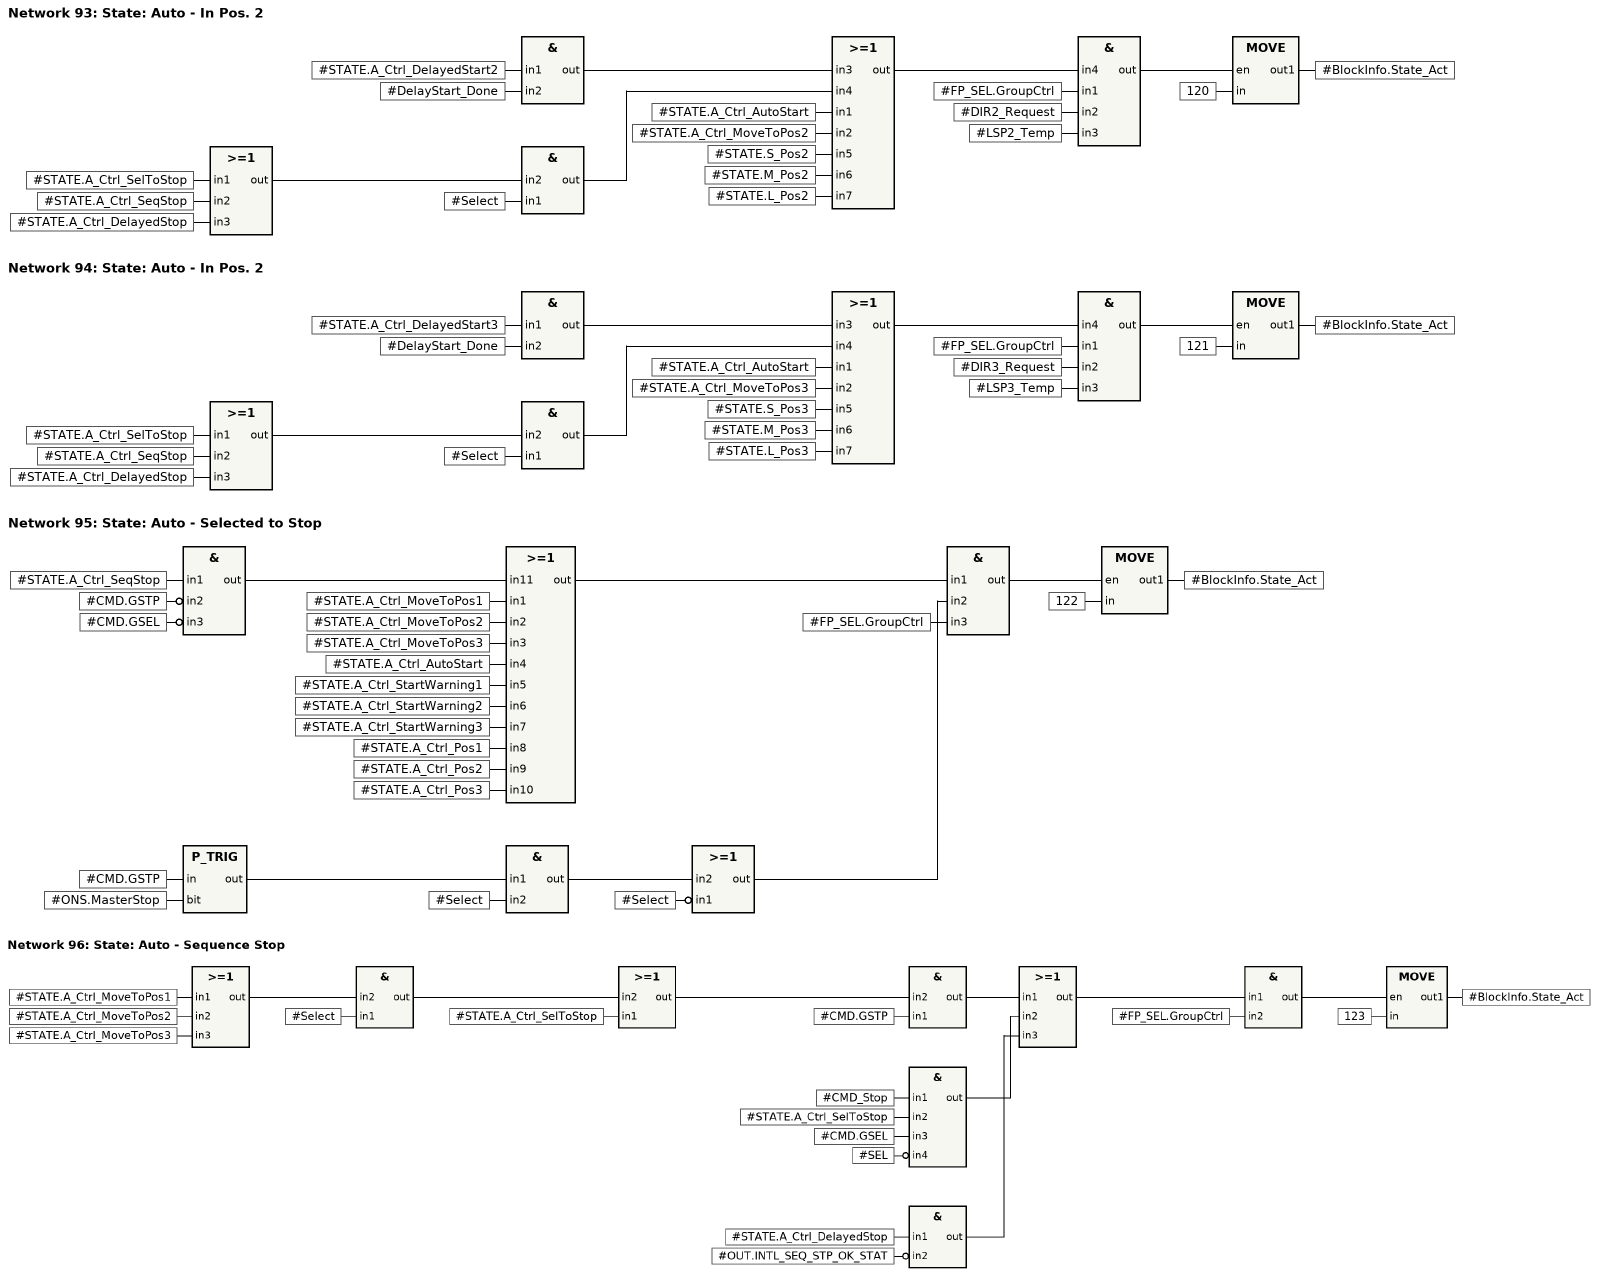
   IF ((#STATE.A_Ctrl_DelayedStart2 AND #DelayStart_Done) OR ((#STATE.A_Ctrl_SelToStop OR #STATE.A_Ctrl_SeqStop OR #STATE.A_Ctrl_DelayedStop) AND #Select) OR #STATE.A_Ctrl_AutoStart OR #STATE.A_Ctrl_MoveToPos2 OR #STATE.S_Pos2 OR #STATE.M_Pos2 OR #STATE.L_Pos2) AND #FP_SEL.GroupCtrl AND #DIR2_Request AND #LSP2_Temp THEN
       #BlockInfo.State_Act := 120;
   END_IF;
END_REGION

REGION Network 94: State: Auto - In Pos. 2
   IF ((#STATE.A_Ctrl_DelayedStart3 AND #DelayStart_Done) OR ((#STATE.A_Ctrl_SelToStop OR #STATE.A_Ctrl_SeqStop OR #STATE.A_Ctrl_DelayedStop) AND #Select) OR #STATE.A_Ctrl_AutoStart OR #STATE.A_Ctrl_MoveToPos3 OR #STATE.S_Pos3 OR #STATE.M_Pos3 OR #STATE.L_Pos3) AND #FP_SEL.GroupCtrl AND #DIR3_Request AND #LSP3_Temp THEN
       #BlockInfo.State_Act := 121;
   END_IF;
END_REGION

REGION Network 95: State: Auto - Selected to Stop
   // Build 004 - 11 Jul 2019 (EXTBOB) : GSEL and A_Ctrl_SeqStop with GSTP condition to move to Selected to Stop state from Seq stop state if group stop timer completes
   #_w1 := #CMD.GSTP AND NOT #ONS.MasterStop;   // rising edge
   #ONS.MasterStop := #CMD.GSTP;
   IF ((#STATE.A_Ctrl_SeqStop AND NOT #CMD.GSTP AND NOT #CMD.GSEL) OR #STATE.A_Ctrl_MoveToPos1 OR #STATE.A_Ctrl_MoveToPos2 OR #STATE.A_Ctrl_MoveToPos3 OR #STATE.A_Ctrl_AutoStart OR #STATE.A_Ctrl_StartWarning1 OR #STATE.A_Ctrl_StartWarning2 OR #STATE.A_Ctrl_StartWarning3 OR #STATE.A_Ctrl_Pos1 OR #STATE.A_Ctrl_Pos2 OR #STATE.A_Ctrl_Pos3) AND ((#_w1 AND #Select) OR NOT #Select) AND #FP_SEL.GroupCtrl THEN
       #BlockInfo.State_Act := 122;
   END_IF;
END_REGION

REGION Network 96: State: Auto - Sequence Stop
   IF (((((#STATE.A_Ctrl_MoveToPos1 OR #STATE.A_Ctrl_MoveToPos2 OR #STATE.A_Ctrl_MoveToPos3) AND #Select) OR #STATE.A_Ctrl_SelToStop) AND #CMD.GSTP) OR (#CMD_Stop AND #STATE.A_Ctrl_SelToStop AND #CMD.GSEL AND NOT #SEL) OR (#STATE.A_Ctrl_DelayedStop AND NOT #OUT.INTL_SEQ_STP_OK_STAT)) AND #FP_SEL.GroupCtrl THEN
       #BlockInfo.State_Act := 123;
   END_IF;
END_REGION

REGION Network 97: State: Auto - Delayed Stop
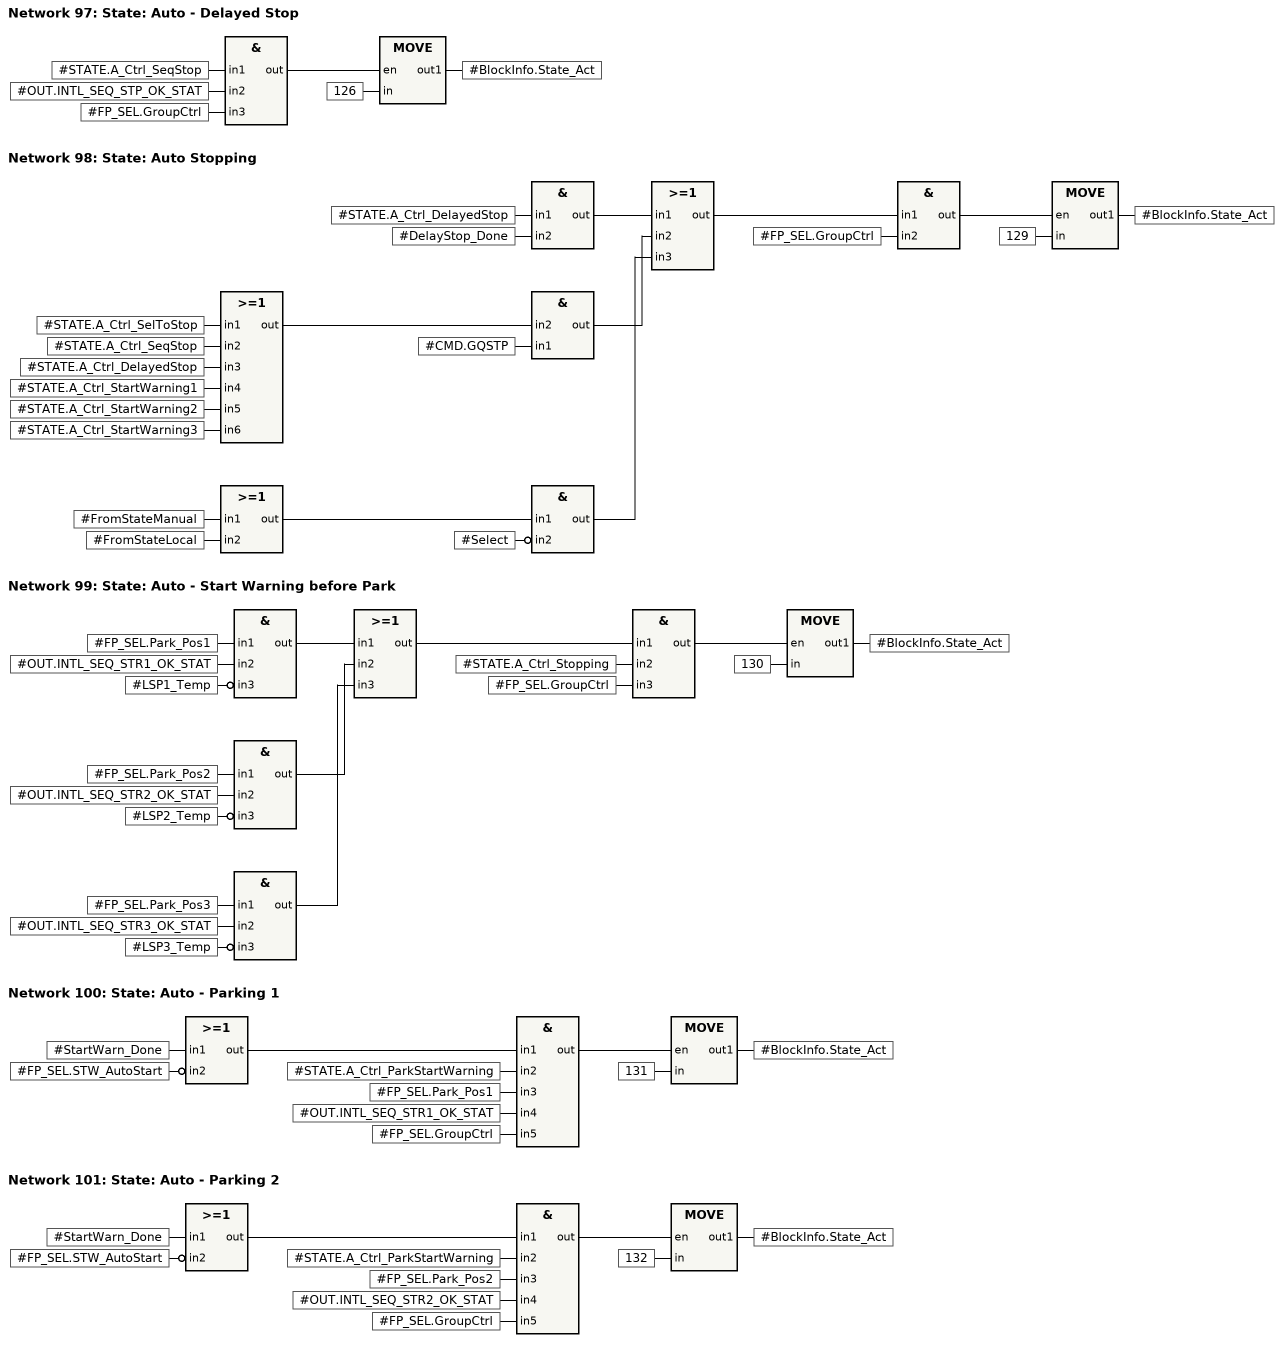
   IF #STATE.A_Ctrl_SeqStop AND #OUT.INTL_SEQ_STP_OK_STAT AND #FP_SEL.GroupCtrl THEN
       #BlockInfo.State_Act := 126;
   END_IF;
END_REGION

REGION Network 98: State: Auto Stopping
   IF ((#STATE.A_Ctrl_DelayedStop AND #DelayStop_Done) OR ((#STATE.A_Ctrl_SelToStop OR #STATE.A_Ctrl_SeqStop OR #STATE.A_Ctrl_DelayedStop OR #STATE.A_Ctrl_StartWarning1 OR #STATE.A_Ctrl_StartWarning2 OR #STATE.A_Ctrl_StartWarning3) AND #CMD.GQSTP) OR ((#FromStateManual OR #FromStateLocal) AND NOT #Select)) AND #FP_SEL.GroupCtrl THEN
       #BlockInfo.State_Act := 129;
   END_IF;
END_REGION

REGION Network 99: State: Auto - Start Warning before Park
   IF ((#FP_SEL.Park_Pos1 AND #OUT.INTL_SEQ_STR1_OK_STAT AND NOT #LSP1_Temp) OR (#FP_SEL.Park_Pos2 AND #OUT.INTL_SEQ_STR2_OK_STAT AND NOT #LSP2_Temp) OR (#FP_SEL.Park_Pos3 AND #OUT.INTL_SEQ_STR3_OK_STAT AND NOT #LSP3_Temp)) AND #STATE.A_Ctrl_Stopping AND #FP_SEL.GroupCtrl THEN
       #BlockInfo.State_Act := 130;
   END_IF;
END_REGION

REGION Network 100: State: Auto - Parking 1
   IF (#StartWarn_Done OR NOT #FP_SEL.STW_AutoStart) AND #STATE.A_Ctrl_ParkStartWarning AND #FP_SEL.Park_Pos1 AND #OUT.INTL_SEQ_STR1_OK_STAT AND #FP_SEL.GroupCtrl THEN
       #BlockInfo.State_Act := 131;
   END_IF;
END_REGION

REGION Network 101: State: Auto - Parking 2
   IF (#StartWarn_Done OR NOT #FP_SEL.STW_AutoStart) AND #STATE.A_Ctrl_ParkStartWarning AND #FP_SEL.Park_Pos2 AND #OUT.INTL_SEQ_STR2_OK_STAT AND #FP_SEL.GroupCtrl THEN
       #BlockInfo.State_Act := 132;
   END_IF;
END_REGION

REGION Network 102: State: Auto - Parking 3
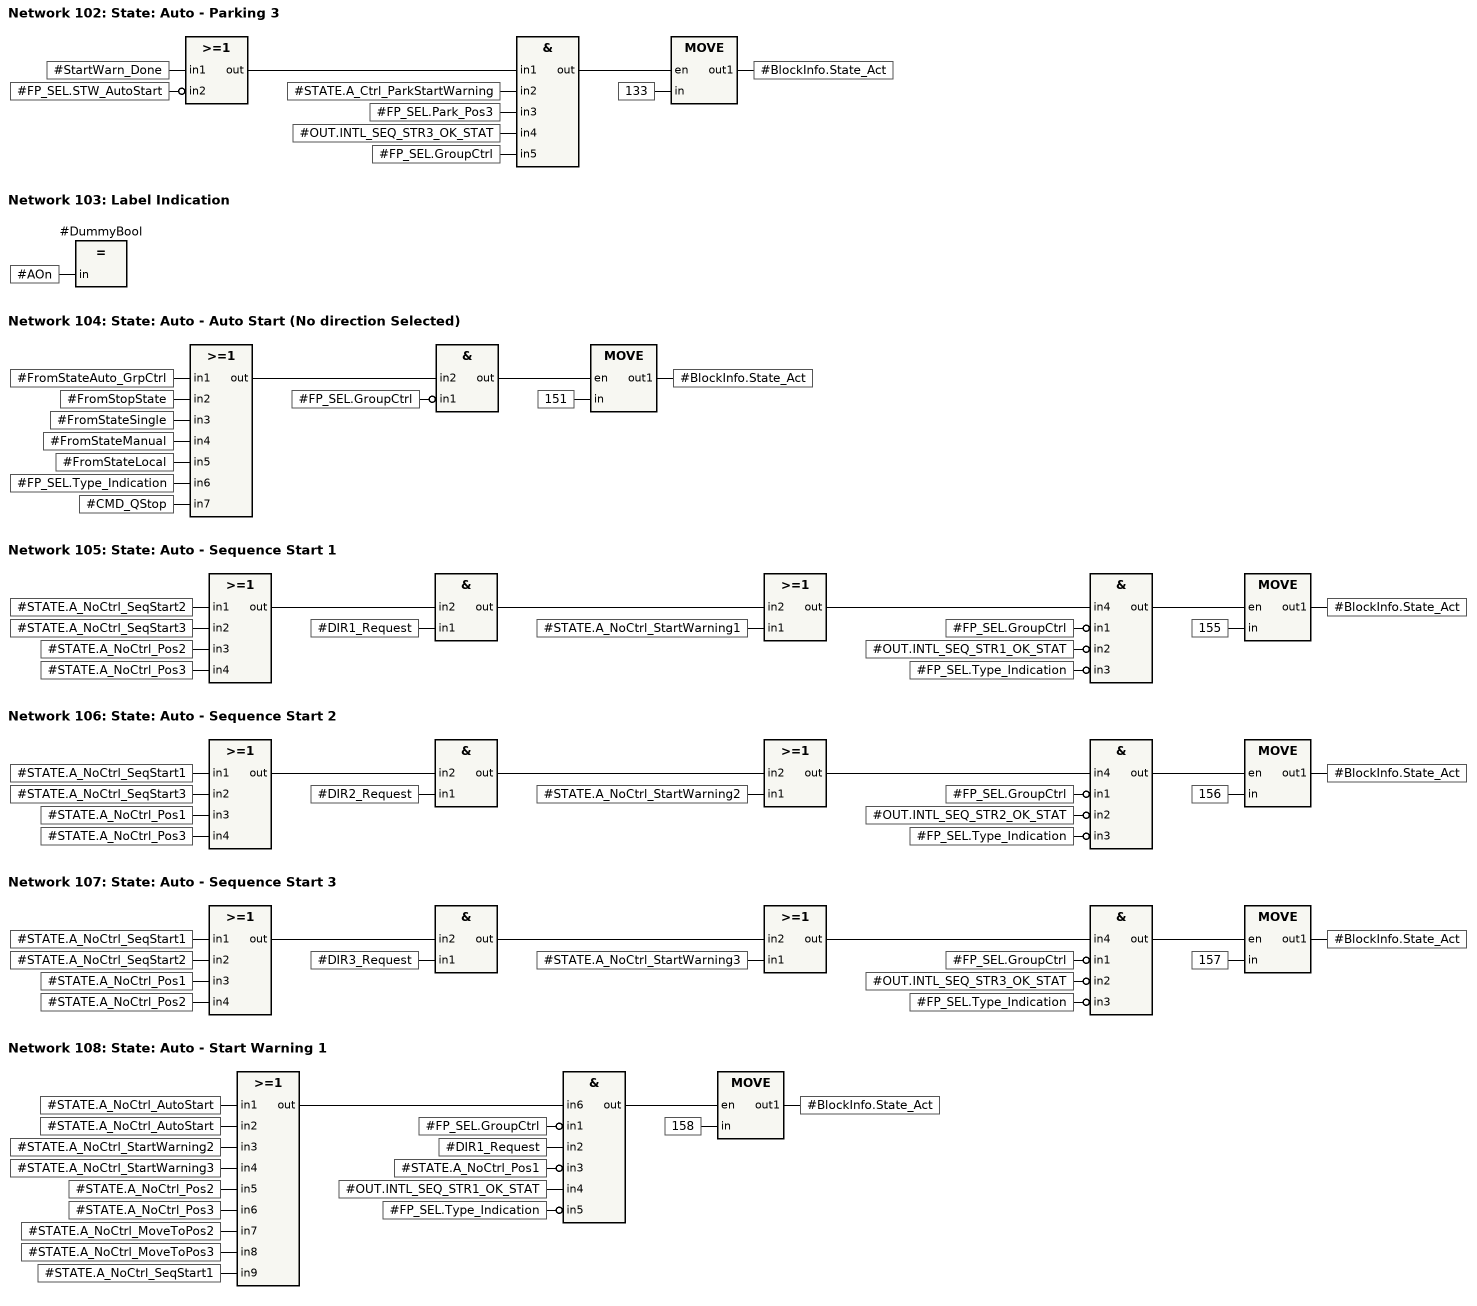
   IF (#StartWarn_Done OR NOT #FP_SEL.STW_AutoStart) AND #STATE.A_Ctrl_ParkStartWarning AND #FP_SEL.Park_Pos3 AND #OUT.INTL_SEQ_STR3_OK_STAT AND #FP_SEL.GroupCtrl THEN
       #BlockInfo.State_Act := 133;
   END_IF;
END_REGION

REGION Network 103: Label Indication
   INDC:
   #DummyBool := #AOn;
END_REGION

REGION Network 104: State: Auto - Auto Start (No direction Selected)
   IF (#FromStateAuto_GrpCtrl OR #FromStopState OR #FromStateSingle OR #FromStateManual OR #FromStateLocal OR #FP_SEL.Type_Indication OR #CMD_QStop) AND NOT #FP_SEL.GroupCtrl THEN
       #BlockInfo.State_Act := 151;
   END_IF;
END_REGION

REGION Network 105: State: Auto - Sequence Start 1
   IF (((#STATE.A_NoCtrl_SeqStart2 OR #STATE.A_NoCtrl_SeqStart3 OR #STATE.A_NoCtrl_Pos2 OR #STATE.A_NoCtrl_Pos3) AND #DIR1_Request) OR #STATE.A_NoCtrl_StartWarning1) AND NOT #FP_SEL.GroupCtrl AND NOT #OUT.INTL_SEQ_STR1_OK_STAT AND NOT #FP_SEL.Type_Indication THEN
       #BlockInfo.State_Act := 155;
   END_IF;
END_REGION

REGION Network 106: State: Auto - Sequence Start 2
   IF (((#STATE.A_NoCtrl_SeqStart1 OR #STATE.A_NoCtrl_SeqStart3 OR #STATE.A_NoCtrl_Pos1 OR #STATE.A_NoCtrl_Pos3) AND #DIR2_Request) OR #STATE.A_NoCtrl_StartWarning2) AND NOT #FP_SEL.GroupCtrl AND NOT #OUT.INTL_SEQ_STR2_OK_STAT AND NOT #FP_SEL.Type_Indication THEN
       #BlockInfo.State_Act := 156;
   END_IF;
END_REGION

REGION Network 107: State: Auto - Sequence Start 3
   IF (((#STATE.A_NoCtrl_SeqStart1 OR #STATE.A_NoCtrl_SeqStart2 OR #STATE.A_NoCtrl_Pos1 OR #STATE.A_NoCtrl_Pos2) AND #DIR3_Request) OR #STATE.A_NoCtrl_StartWarning3) AND NOT #FP_SEL.GroupCtrl AND NOT #OUT.INTL_SEQ_STR3_OK_STAT AND NOT #FP_SEL.Type_Indication THEN
       #BlockInfo.State_Act := 157;
   END_IF;
END_REGION

REGION Network 108: State: Auto - Start Warning 1
   IF (#STATE.A_NoCtrl_AutoStart OR #STATE.A_NoCtrl_AutoStart OR #STATE.A_NoCtrl_StartWarning2 OR #STATE.A_NoCtrl_StartWarning3 OR #STATE.A_NoCtrl_Pos2 OR #STATE.A_NoCtrl_Pos3 OR #STATE.A_NoCtrl_MoveToPos2 OR #STATE.A_NoCtrl_MoveToPos3 OR #STATE.A_NoCtrl_SeqStart1) AND NOT #FP_SEL.GroupCtrl AND #DIR1_Request AND NOT #STATE.A_NoCtrl_Pos1 AND #OUT.INTL_SEQ_STR1_OK_STAT AND NOT #FP_SEL.Type_Indication THEN
       #BlockInfo.State_Act := 158;
   END_IF;
END_REGION

REGION Network 109: State: Auto - Start Warning 2
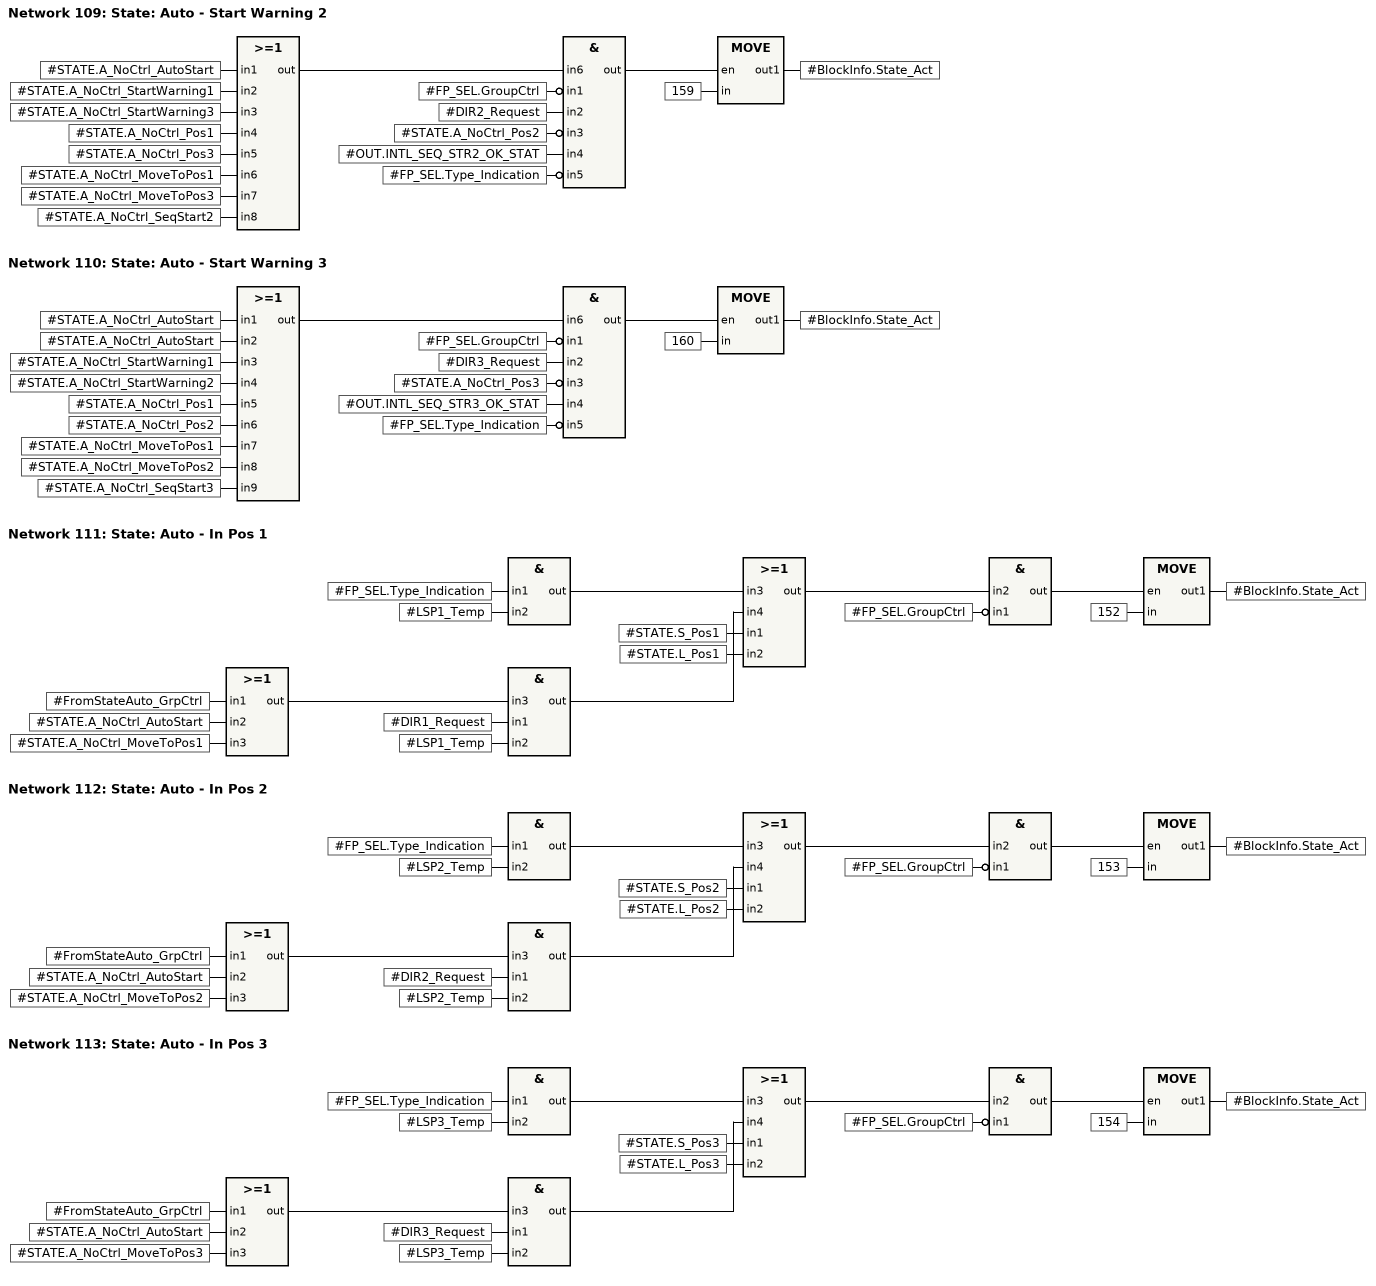
   IF (#STATE.A_NoCtrl_AutoStart OR #STATE.A_NoCtrl_StartWarning1 OR #STATE.A_NoCtrl_StartWarning3 OR #STATE.A_NoCtrl_Pos1 OR #STATE.A_NoCtrl_Pos3 OR #STATE.A_NoCtrl_MoveToPos1 OR #STATE.A_NoCtrl_MoveToPos3 OR #STATE.A_NoCtrl_SeqStart2) AND NOT #FP_SEL.GroupCtrl AND #DIR2_Request AND NOT #STATE.A_NoCtrl_Pos2 AND #OUT.INTL_SEQ_STR2_OK_STAT AND NOT #FP_SEL.Type_Indication THEN
       #BlockInfo.State_Act := 159;
   END_IF;
END_REGION

REGION Network 110: State: Auto - Start Warning 3
   IF (#STATE.A_NoCtrl_AutoStart OR #STATE.A_NoCtrl_AutoStart OR #STATE.A_NoCtrl_StartWarning1 OR #STATE.A_NoCtrl_StartWarning2 OR #STATE.A_NoCtrl_Pos1 OR #STATE.A_NoCtrl_Pos2 OR #STATE.A_NoCtrl_MoveToPos1 OR #STATE.A_NoCtrl_MoveToPos2 OR #STATE.A_NoCtrl_SeqStart3) AND NOT #FP_SEL.GroupCtrl AND #DIR3_Request AND NOT #STATE.A_NoCtrl_Pos3 AND #OUT.INTL_SEQ_STR3_OK_STAT AND NOT #FP_SEL.Type_Indication THEN
       #BlockInfo.State_Act := 160;
   END_IF;
END_REGION

REGION Network 111: State: Auto - In Pos 1
   IF ((#FP_SEL.Type_Indication AND #LSP1_Temp) OR ((#FromStateAuto_GrpCtrl OR #STATE.A_NoCtrl_AutoStart OR #STATE.A_NoCtrl_MoveToPos1) AND #DIR1_Request AND #LSP1_Temp) OR #STATE.S_Pos1 OR #STATE.L_Pos1) AND NOT #FP_SEL.GroupCtrl THEN
       #BlockInfo.State_Act := 152;
   END_IF;
END_REGION

REGION Network 112: State: Auto - In Pos 2
   IF ((#FP_SEL.Type_Indication AND #LSP2_Temp) OR ((#FromStateAuto_GrpCtrl OR #STATE.A_NoCtrl_AutoStart OR #STATE.A_NoCtrl_MoveToPos2) AND #DIR2_Request AND #LSP2_Temp) OR #STATE.S_Pos2 OR #STATE.L_Pos2) AND NOT #FP_SEL.GroupCtrl THEN
       #BlockInfo.State_Act := 153;
   END_IF;
END_REGION

REGION Network 113: State: Auto - In Pos 3
   IF ((#FP_SEL.Type_Indication AND #LSP3_Temp) OR ((#FromStateAuto_GrpCtrl OR #STATE.A_NoCtrl_AutoStart OR #STATE.A_NoCtrl_MoveToPos3) AND #DIR3_Request AND #LSP3_Temp) OR #STATE.S_Pos3 OR #STATE.L_Pos3) AND NOT #FP_SEL.GroupCtrl THEN
       #BlockInfo.State_Act := 154;
   END_IF;
END_REGION

REGION Network 114: State: Auto - Running 1
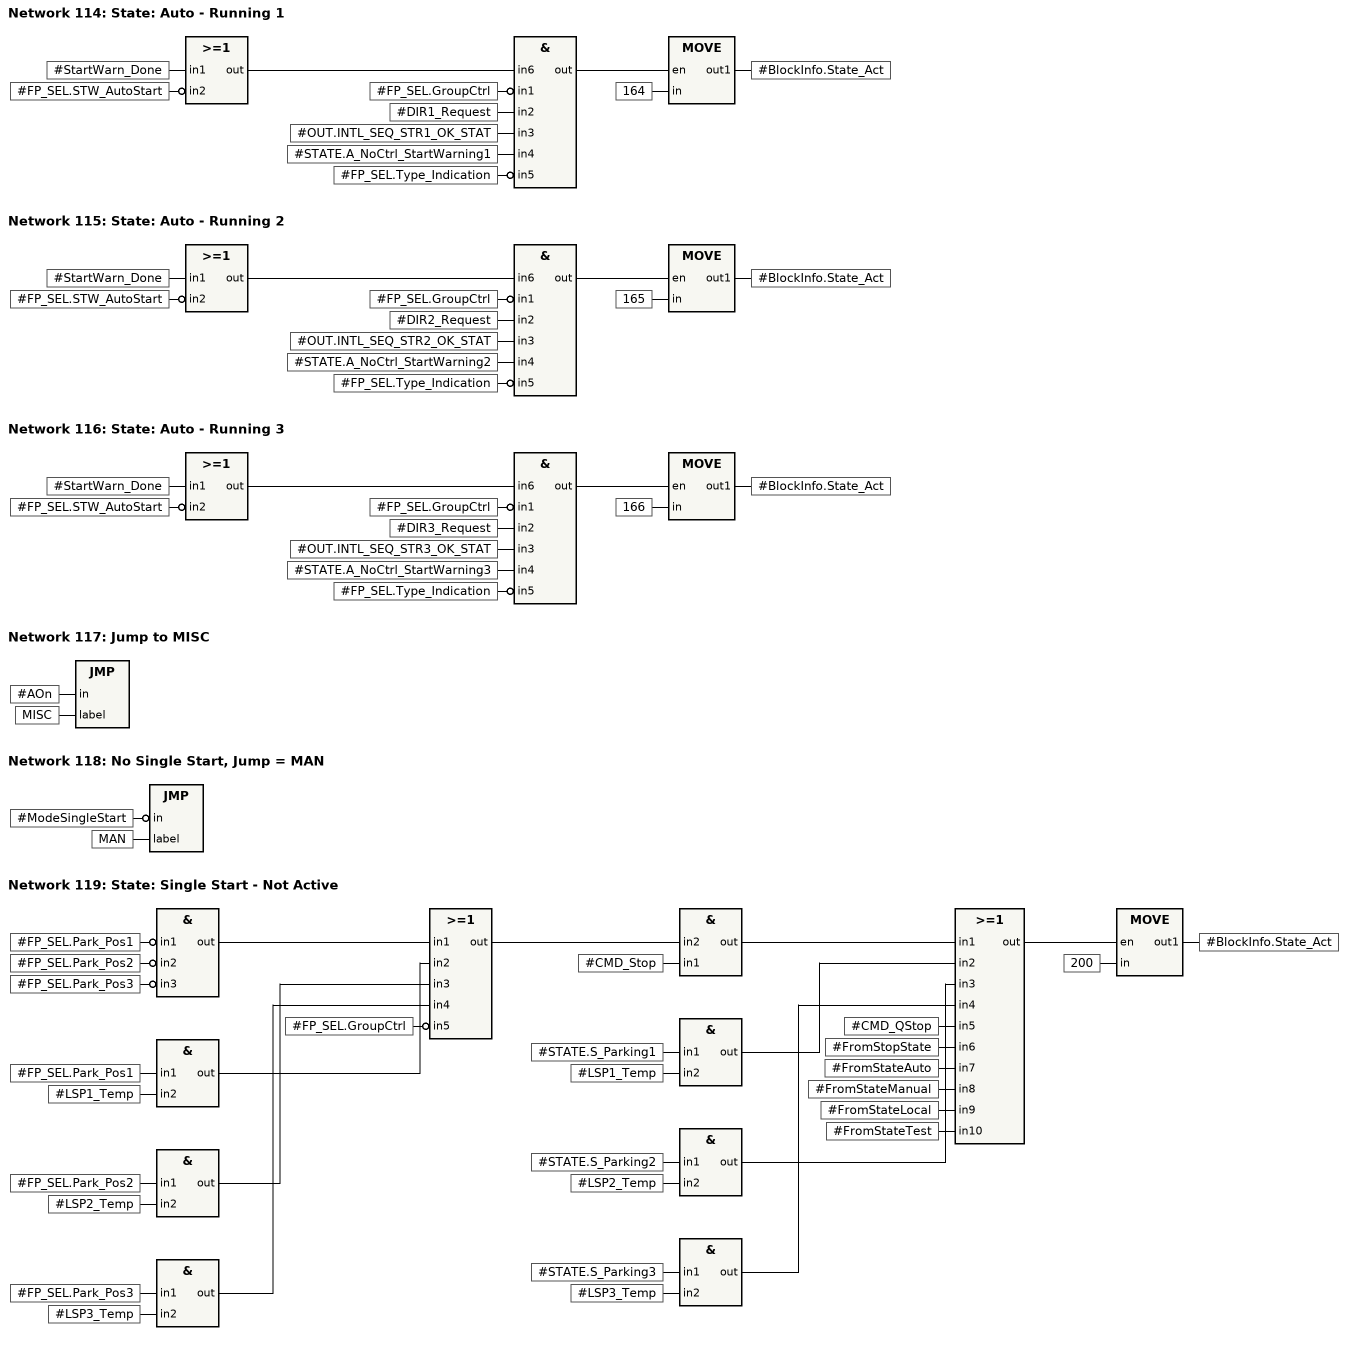
   IF (#StartWarn_Done OR NOT #FP_SEL.STW_AutoStart) AND NOT #FP_SEL.GroupCtrl AND #DIR1_Request AND #OUT.INTL_SEQ_STR1_OK_STAT AND #STATE.A_NoCtrl_StartWarning1 AND NOT #FP_SEL.Type_Indication THEN
       #BlockInfo.State_Act := 164;
   END_IF;
END_REGION

REGION Network 115: State: Auto - Running 2
   IF (#StartWarn_Done OR NOT #FP_SEL.STW_AutoStart) AND NOT #FP_SEL.GroupCtrl AND #DIR2_Request AND #OUT.INTL_SEQ_STR2_OK_STAT AND #STATE.A_NoCtrl_StartWarning2 AND NOT #FP_SEL.Type_Indication THEN
       #BlockInfo.State_Act := 165;
   END_IF;
END_REGION

REGION Network 116: State: Auto - Running 3
   IF (#StartWarn_Done OR NOT #FP_SEL.STW_AutoStart) AND NOT #FP_SEL.GroupCtrl AND #DIR3_Request AND #OUT.INTL_SEQ_STR3_OK_STAT AND #STATE.A_NoCtrl_StartWarning3 AND NOT #FP_SEL.Type_Indication THEN
       #BlockInfo.State_Act := 166;
   END_IF;
END_REGION

REGION Network 117: Jump to MISC
   IF #AOn THEN GOTO MISC; END_IF;
END_REGION

REGION Network 118: No Single Start, Jump = MAN
   SS1:
   IF NOT #ModeSingleStart THEN GOTO MAN; END_IF;
END_REGION

REGION Network 119: State: Single Start - Not Active
   IF (((NOT #FP_SEL.Park_Pos1 AND NOT #FP_SEL.Park_Pos2 AND NOT #FP_SEL.Park_Pos3) OR (#FP_SEL.Park_Pos1 AND #LSP1_Temp) OR (#FP_SEL.Park_Pos2 AND #LSP2_Temp) OR (#FP_SEL.Park_Pos3 AND #LSP3_Temp) OR NOT #FP_SEL.GroupCtrl) AND #CMD_Stop) OR (#STATE.S_Parking1 AND #LSP1_Temp) OR (#STATE.S_Parking2 AND #LSP2_Temp) OR (#STATE.S_Parking3 AND #LSP3_Temp) OR #CMD_QStop OR #FromStopState OR #FromStateAuto OR #FromStateManual OR #FromStateLocal OR #FromStateTest THEN
       #BlockInfo.State_Act := 200;
   END_IF;
END_REGION

REGION Network 120: State: Single Start - Start Warning 1
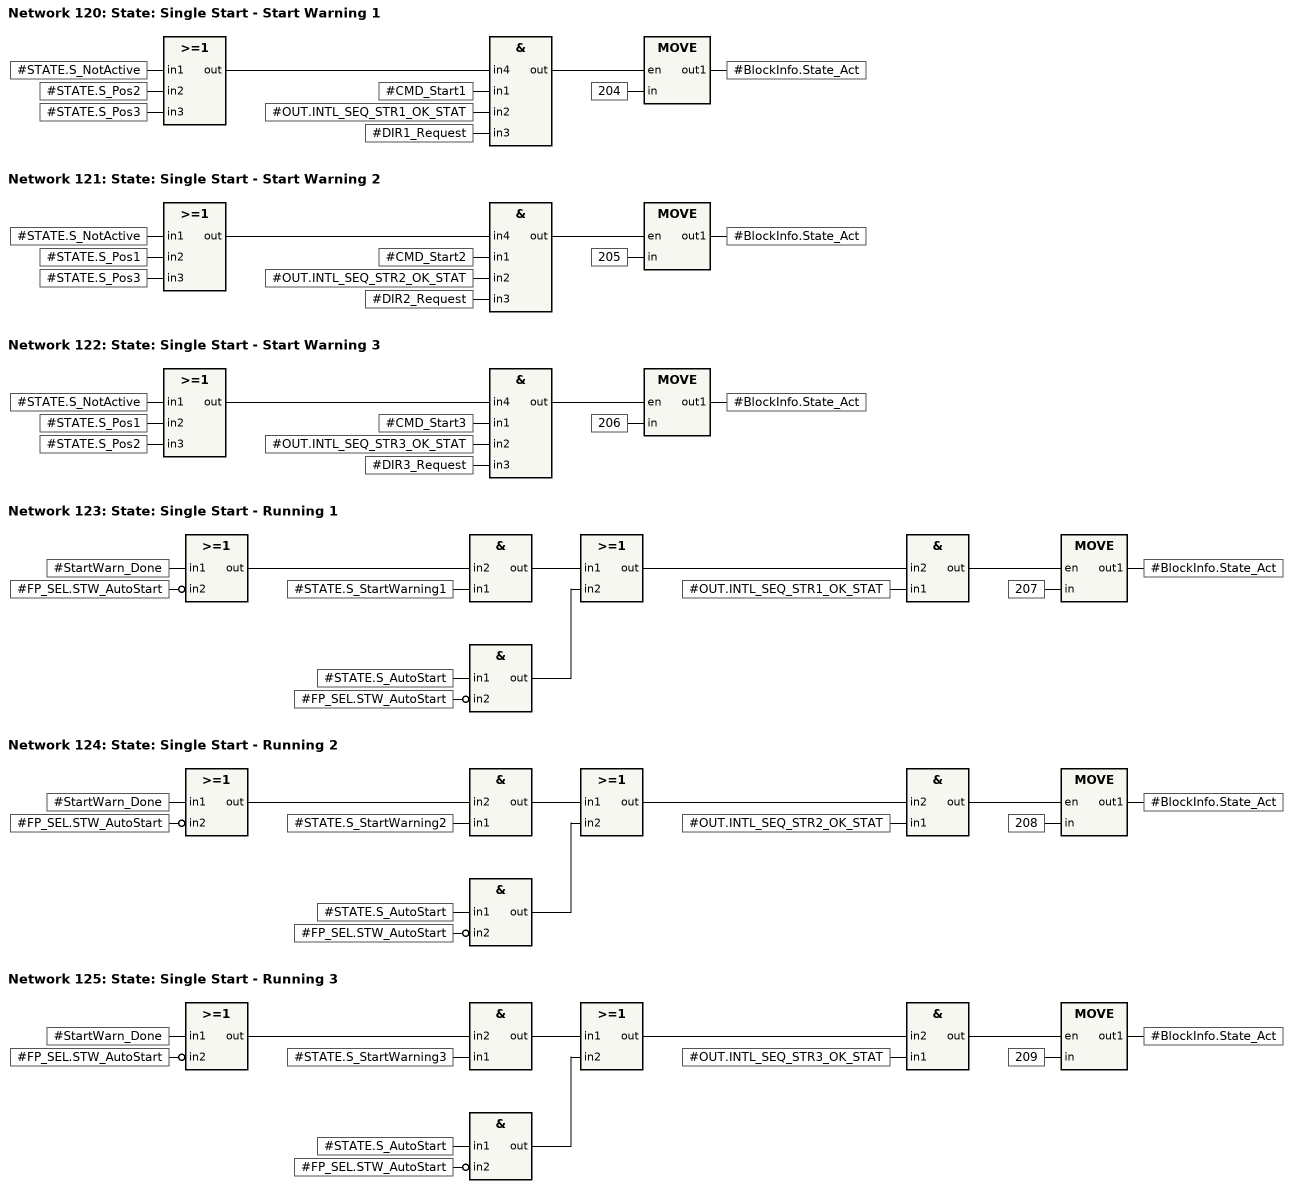
   IF (#STATE.S_NotActive OR #STATE.S_Pos2 OR #STATE.S_Pos3) AND #CMD_Start1 AND #OUT.INTL_SEQ_STR1_OK_STAT AND #DIR1_Request THEN
       #BlockInfo.State_Act := 204;
   END_IF;
END_REGION

REGION Network 121: State: Single Start - Start Warning 2
   IF (#STATE.S_NotActive OR #STATE.S_Pos1 OR #STATE.S_Pos3) AND #CMD_Start2 AND #OUT.INTL_SEQ_STR2_OK_STAT AND #DIR2_Request THEN
       #BlockInfo.State_Act := 205;
   END_IF;
END_REGION

REGION Network 122: State: Single Start - Start Warning 3
   IF (#STATE.S_NotActive OR #STATE.S_Pos1 OR #STATE.S_Pos2) AND #CMD_Start3 AND #OUT.INTL_SEQ_STR3_OK_STAT AND #DIR3_Request THEN
       #BlockInfo.State_Act := 206;
   END_IF;
END_REGION

REGION Network 123: State: Single Start - Running 1
   IF (((#StartWarn_Done OR NOT #FP_SEL.STW_AutoStart) AND #STATE.S_StartWarning1) OR (#STATE.S_AutoStart AND NOT #FP_SEL.STW_AutoStart)) AND #OUT.INTL_SEQ_STR1_OK_STAT THEN
       #BlockInfo.State_Act := 207;
   END_IF;
END_REGION

REGION Network 124: State: Single Start - Running 2
   IF (((#StartWarn_Done OR NOT #FP_SEL.STW_AutoStart) AND #STATE.S_StartWarning2) OR (#STATE.S_AutoStart AND NOT #FP_SEL.STW_AutoStart)) AND #OUT.INTL_SEQ_STR2_OK_STAT THEN
       #BlockInfo.State_Act := 208;
   END_IF;
END_REGION

REGION Network 125: State: Single Start - Running 3
   IF (((#StartWarn_Done OR NOT #FP_SEL.STW_AutoStart) AND #STATE.S_StartWarning3) OR (#STATE.S_AutoStart AND NOT #FP_SEL.STW_AutoStart)) AND #OUT.INTL_SEQ_STR3_OK_STAT THEN
       #BlockInfo.State_Act := 209;
   END_IF;
END_REGION

REGION Network 126: State: Single Start - Auto Start (No Direction Selected)
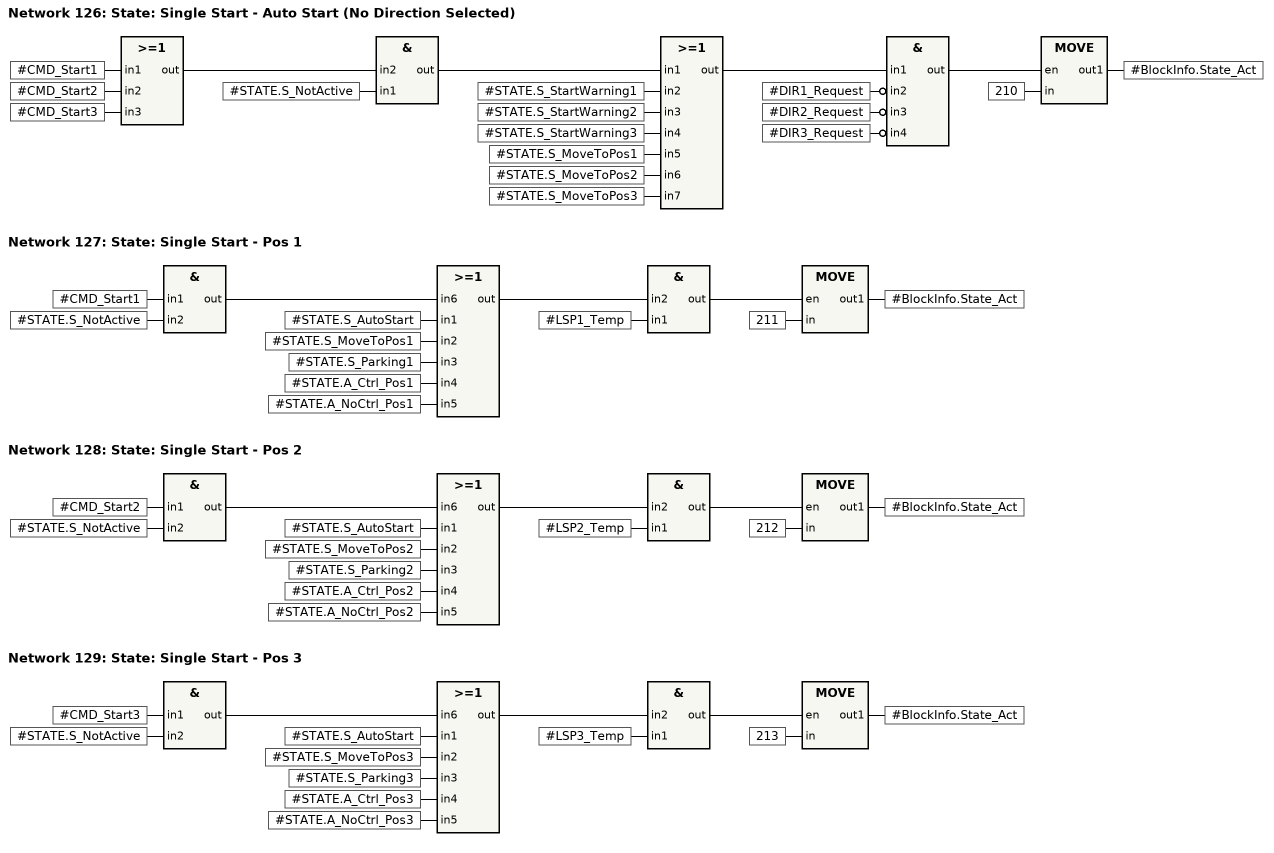
   IF (((#CMD_Start1 OR #CMD_Start2 OR #CMD_Start3) AND #STATE.S_NotActive) OR #STATE.S_StartWarning1 OR #STATE.S_StartWarning2 OR #STATE.S_StartWarning3 OR #STATE.S_MoveToPos1 OR #STATE.S_MoveToPos2 OR #STATE.S_MoveToPos3) AND NOT #DIR1_Request AND NOT #DIR2_Request AND NOT #DIR3_Request THEN
       #BlockInfo.State_Act := 210;
   END_IF;
END_REGION

REGION Network 127: State: Single Start - Pos 1
   IF ((#CMD_Start1 AND #STATE.S_NotActive) OR #STATE.S_AutoStart OR #STATE.S_MoveToPos1 OR #STATE.S_Parking1 OR #STATE.A_Ctrl_Pos1 OR #STATE.A_NoCtrl_Pos1) AND #LSP1_Temp THEN
       #BlockInfo.State_Act := 211;
   END_IF;
END_REGION

REGION Network 128: State: Single Start - Pos 2
   IF ((#CMD_Start2 AND #STATE.S_NotActive) OR #STATE.S_AutoStart OR #STATE.S_MoveToPos2 OR #STATE.S_Parking2 OR #STATE.A_Ctrl_Pos2 OR #STATE.A_NoCtrl_Pos2) AND #LSP2_Temp THEN
       #BlockInfo.State_Act := 212;
   END_IF;
END_REGION

REGION Network 129: State: Single Start - Pos 3
   IF ((#CMD_Start3 AND #STATE.S_NotActive) OR #STATE.S_AutoStart OR #STATE.S_MoveToPos3 OR #STATE.S_Parking3 OR #STATE.A_Ctrl_Pos3 OR #STATE.A_NoCtrl_Pos3) AND #LSP3_Temp THEN
       #BlockInfo.State_Act := 213;
   END_IF;
END_REGION

REGION Network 130: State: Single Start - Stop
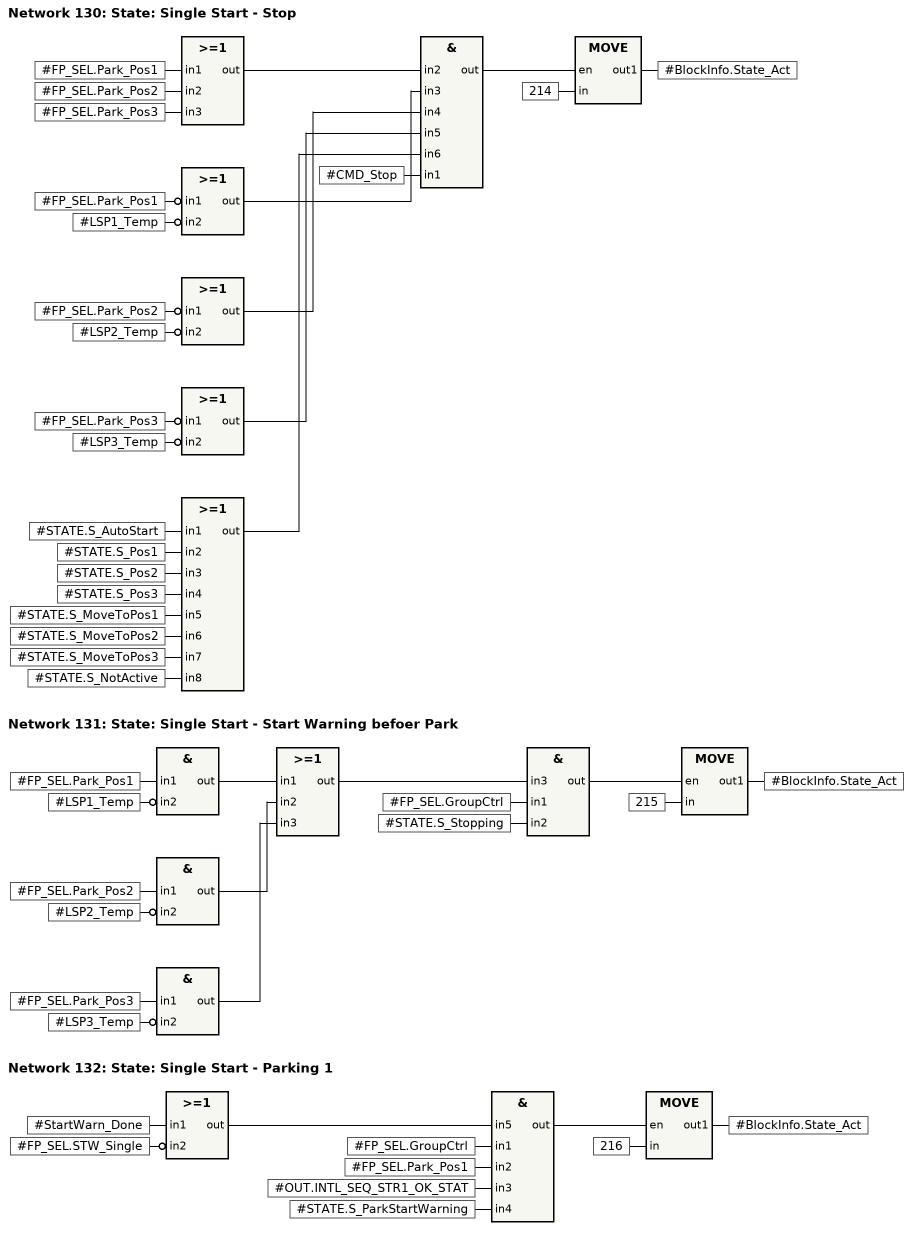
   IF (#FP_SEL.Park_Pos1 OR #FP_SEL.Park_Pos2 OR #FP_SEL.Park_Pos3) AND (NOT #FP_SEL.Park_Pos1 OR NOT #LSP1_Temp) AND (NOT #FP_SEL.Park_Pos2 OR NOT #LSP2_Temp) AND (NOT #FP_SEL.Park_Pos3 OR NOT #LSP3_Temp) AND (#STATE.S_AutoStart OR #STATE.S_Pos1 OR #STATE.S_Pos2 OR #STATE.S_Pos3 OR #STATE.S_MoveToPos1 OR #STATE.S_MoveToPos2 OR #STATE.S_MoveToPos3 OR #STATE.S_NotActive) AND #CMD_Stop THEN
       #BlockInfo.State_Act := 214;
   END_IF;
END_REGION

REGION Network 131: State: Single Start - Start Warning befoer Park
   IF ((#FP_SEL.Park_Pos1 AND NOT #LSP1_Temp) OR (#FP_SEL.Park_Pos2 AND NOT #LSP2_Temp) OR (#FP_SEL.Park_Pos3 AND NOT #LSP3_Temp)) AND #FP_SEL.GroupCtrl AND #STATE.S_Stopping THEN
       #BlockInfo.State_Act := 215;
   END_IF;
END_REGION

REGION Network 132: State: Single Start - Parking 1
   IF (#StartWarn_Done OR NOT #FP_SEL.STW_Single) AND #FP_SEL.GroupCtrl AND #FP_SEL.Park_Pos1 AND #OUT.INTL_SEQ_STR1_OK_STAT AND #STATE.S_ParkStartWarning THEN
       #BlockInfo.State_Act := 216;
   END_IF;
END_REGION

REGION Network 133: State: Single Start - Parking 2
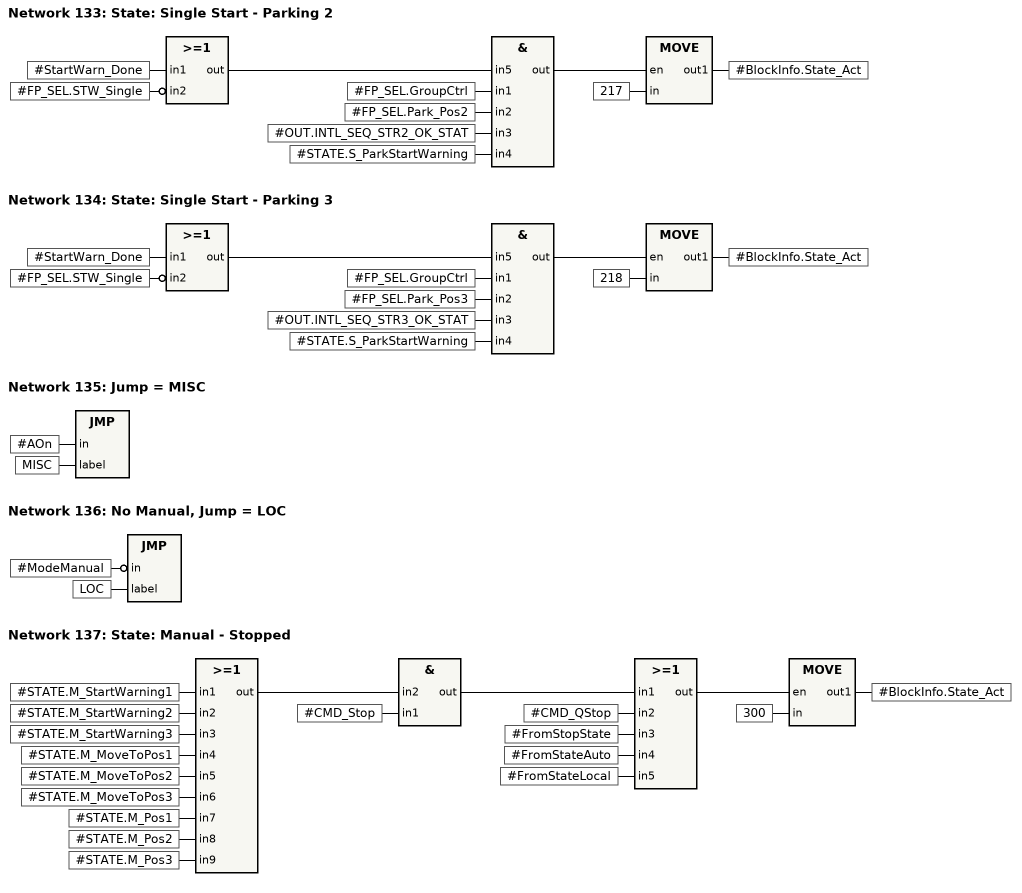
   IF (#StartWarn_Done OR NOT #FP_SEL.STW_Single) AND #FP_SEL.GroupCtrl AND #FP_SEL.Park_Pos2 AND #OUT.INTL_SEQ_STR2_OK_STAT AND #STATE.S_ParkStartWarning THEN
       #BlockInfo.State_Act := 217;
   END_IF;
END_REGION

REGION Network 134: State: Single Start - Parking 3
   IF (#StartWarn_Done OR NOT #FP_SEL.STW_Single) AND #FP_SEL.GroupCtrl AND #FP_SEL.Park_Pos3 AND #OUT.INTL_SEQ_STR3_OK_STAT AND #STATE.S_ParkStartWarning THEN
       #BlockInfo.State_Act := 218;
   END_IF;
END_REGION

REGION Network 135: Jump = MISC
   IF #AOn THEN GOTO MISC; END_IF;
END_REGION

REGION Network 136: No Manual, Jump = LOC
   MAN:
   IF NOT #ModeManual THEN GOTO LOC; END_IF;
END_REGION

REGION Network 137: State: Manual - Stopped
   IF ((#STATE.M_StartWarning1 OR #STATE.M_StartWarning2 OR #STATE.M_StartWarning3 OR #STATE.M_MoveToPos1 OR #STATE.M_MoveToPos2 OR #STATE.M_MoveToPos3 OR #STATE.M_Pos1 OR #STATE.M_Pos2 OR #STATE.M_Pos3) AND #CMD_Stop) OR #CMD_QStop OR #FromStopState OR #FromStateAuto OR #FromStateLocal THEN
       #BlockInfo.State_Act := 300;
   END_IF;
END_REGION

REGION Network 138: State: Manual - Active (Autostart)
   // Build 006 - 21.Feb.2022 (SURAM-IN) FP_CMD.Start1,  FP_CMD.Start2,  FP_CMD.Start3 and FP_SEL.INCH_Man logic added for Inching in Manual Mode
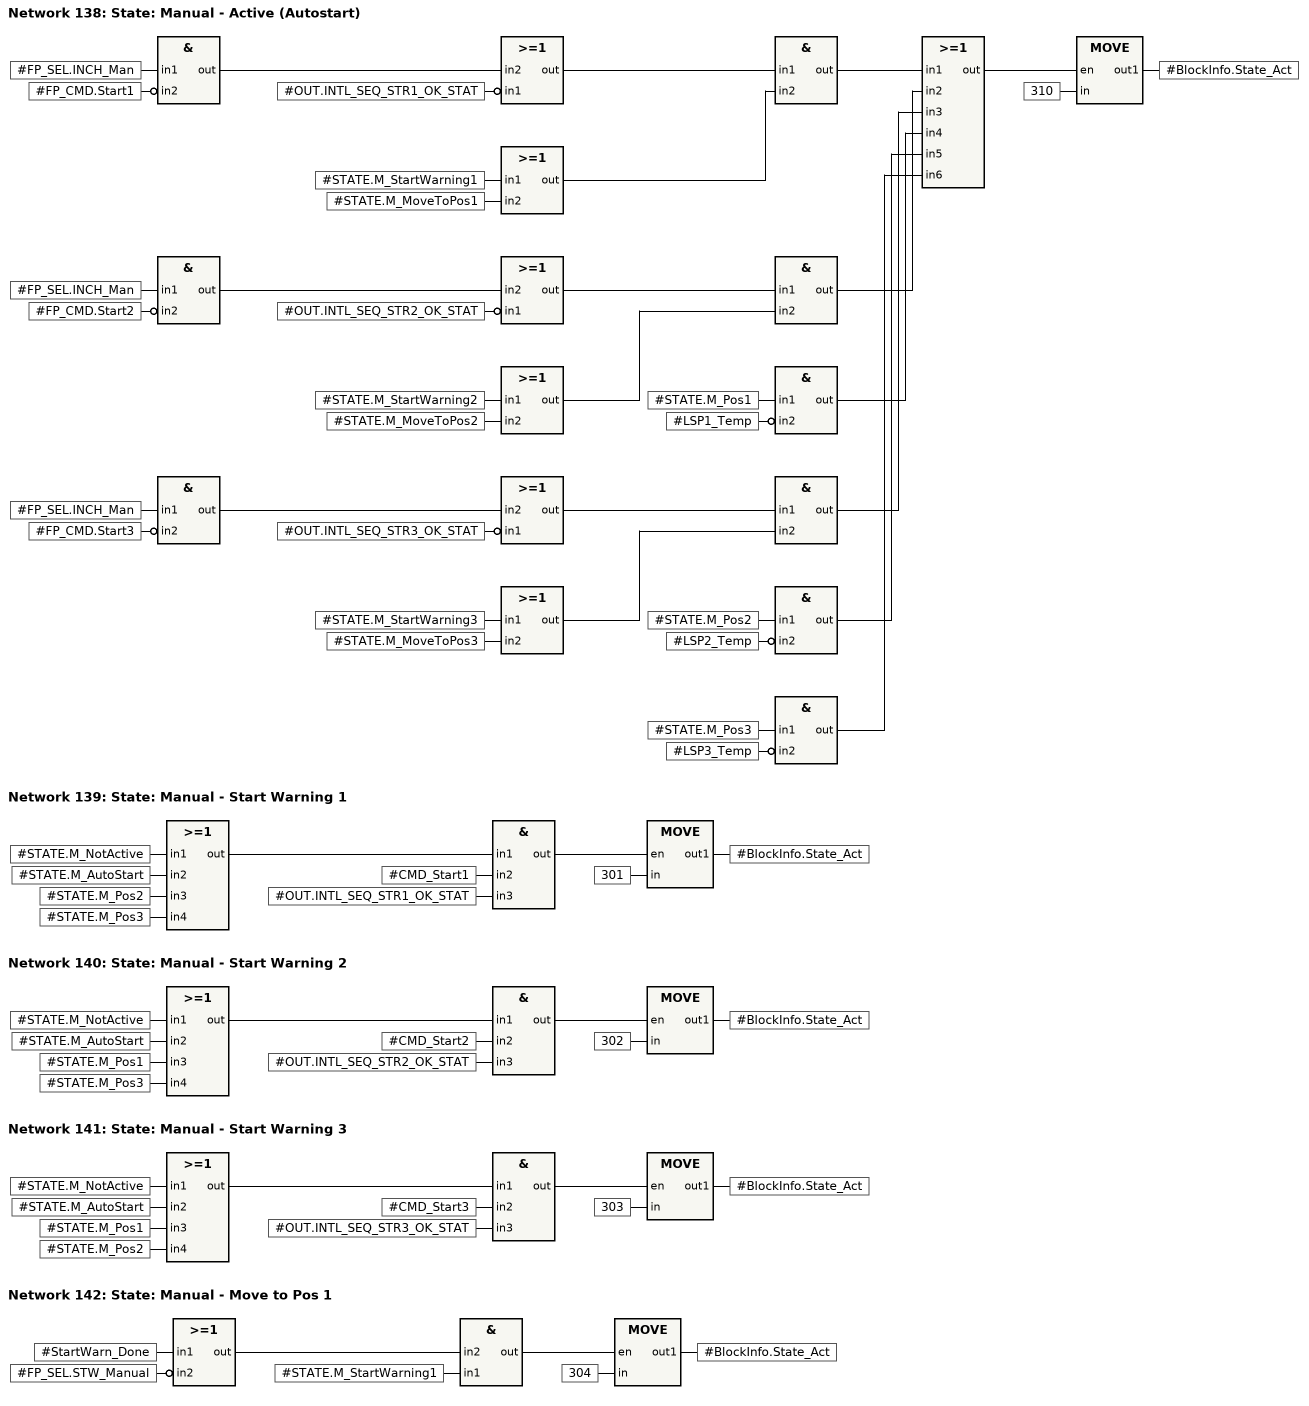
   IF (((#FP_SEL.INCH_Man AND NOT #FP_CMD.Start1) OR NOT #OUT.INTL_SEQ_STR1_OK_STAT) AND (#STATE.M_StartWarning1 OR #STATE.M_MoveToPos1)) OR (((#FP_SEL.INCH_Man AND NOT #FP_CMD.Start2) OR NOT #OUT.INTL_SEQ_STR2_OK_STAT) AND (#STATE.M_StartWarning2 OR #STATE.M_MoveToPos2)) OR (((#FP_SEL.INCH_Man AND NOT #FP_CMD.Start3) OR NOT #OUT.INTL_SEQ_STR3_OK_STAT) AND (#STATE.M_StartWarning3 OR #STATE.M_MoveToPos3)) OR (#STATE.M_Pos1 AND NOT #LSP1_Temp) OR (#STATE.M_Pos2 AND NOT #LSP2_Temp) OR (#STATE.M_Pos3 AND NOT #LSP3_Temp) THEN
       #BlockInfo.State_Act := 310;
   END_IF;
END_REGION

REGION Network 139: State: Manual - Start Warning 1
   IF (#STATE.M_NotActive OR #STATE.M_AutoStart OR #STATE.M_Pos2 OR #STATE.M_Pos3) AND #CMD_Start1 AND #OUT.INTL_SEQ_STR1_OK_STAT THEN
       #BlockInfo.State_Act := 301;
   END_IF;
END_REGION

REGION Network 140: State: Manual - Start Warning 2
   IF (#STATE.M_NotActive OR #STATE.M_AutoStart OR #STATE.M_Pos1 OR #STATE.M_Pos3) AND #CMD_Start2 AND #OUT.INTL_SEQ_STR2_OK_STAT THEN
       #BlockInfo.State_Act := 302;
   END_IF;
END_REGION

REGION Network 141: State: Manual - Start Warning 3
   IF (#STATE.M_NotActive OR #STATE.M_AutoStart OR #STATE.M_Pos1 OR #STATE.M_Pos2) AND #CMD_Start3 AND #OUT.INTL_SEQ_STR3_OK_STAT THEN
       #BlockInfo.State_Act := 303;
   END_IF;
END_REGION

REGION Network 142: State: Manual - Move to Pos 1
   IF (#StartWarn_Done OR NOT #FP_SEL.STW_Manual) AND #STATE.M_StartWarning1 THEN
       #BlockInfo.State_Act := 304;
   END_IF;
END_REGION

REGION Network 143: State: Manual - Move to Pos 2
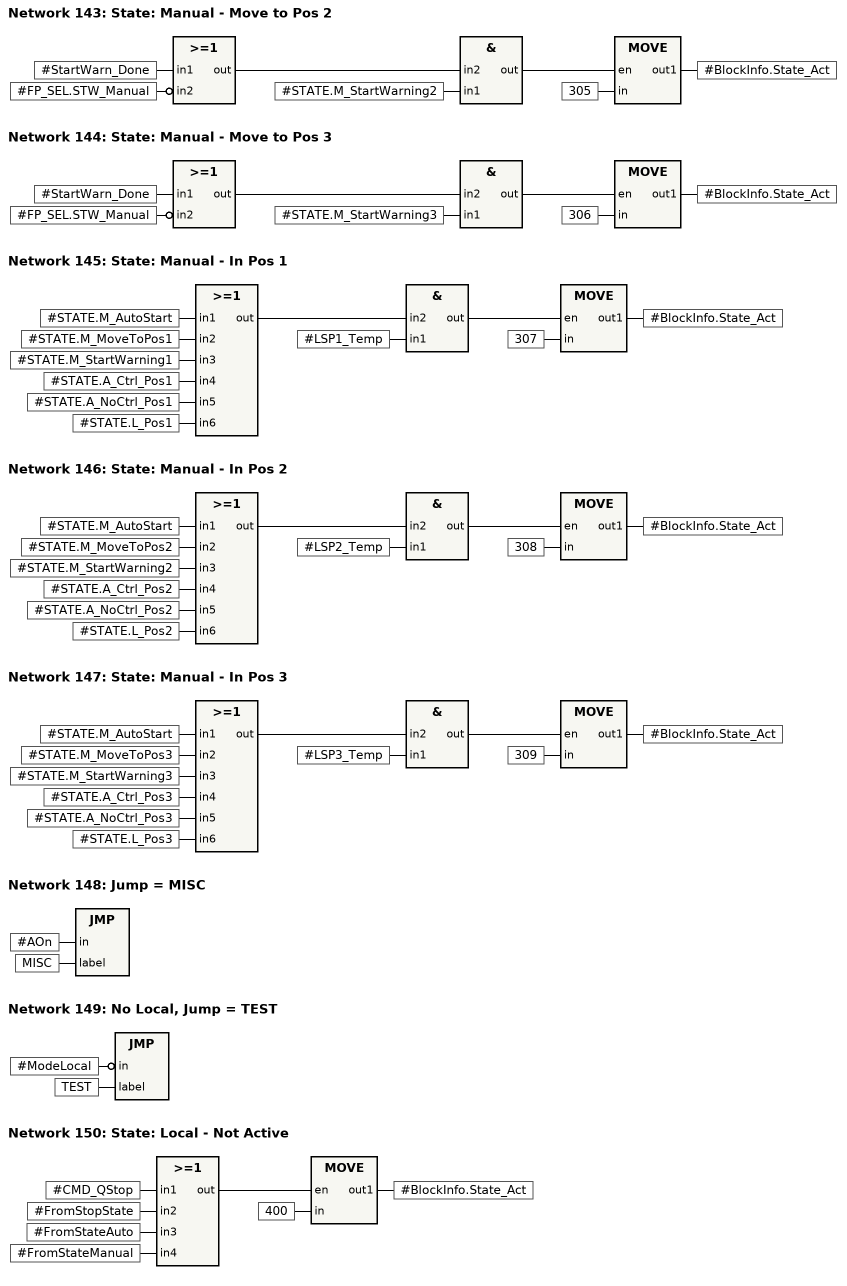
   IF (#StartWarn_Done OR NOT #FP_SEL.STW_Manual) AND #STATE.M_StartWarning2 THEN
       #BlockInfo.State_Act := 305;
   END_IF;
END_REGION

REGION Network 144: State: Manual - Move to Pos 3
   IF (#StartWarn_Done OR NOT #FP_SEL.STW_Manual) AND #STATE.M_StartWarning3 THEN
       #BlockInfo.State_Act := 306;
   END_IF;
END_REGION

REGION Network 145: State: Manual - In Pos 1
   IF (#STATE.M_AutoStart OR #STATE.M_MoveToPos1 OR #STATE.M_StartWarning1 OR #STATE.A_Ctrl_Pos1 OR #STATE.A_NoCtrl_Pos1 OR #STATE.L_Pos1) AND #LSP1_Temp THEN
       #BlockInfo.State_Act := 307;
   END_IF;
END_REGION

REGION Network 146: State: Manual - In Pos 2
   IF (#STATE.M_AutoStart OR #STATE.M_MoveToPos2 OR #STATE.M_StartWarning2 OR #STATE.A_Ctrl_Pos2 OR #STATE.A_NoCtrl_Pos2 OR #STATE.L_Pos2) AND #LSP2_Temp THEN
       #BlockInfo.State_Act := 308;
   END_IF;
END_REGION

REGION Network 147: State: Manual - In Pos 3
   IF (#STATE.M_AutoStart OR #STATE.M_MoveToPos3 OR #STATE.M_StartWarning3 OR #STATE.A_Ctrl_Pos3 OR #STATE.A_NoCtrl_Pos3 OR #STATE.L_Pos3) AND #LSP3_Temp THEN
       #BlockInfo.State_Act := 309;
   END_IF;
END_REGION

REGION Network 148: Jump = MISC
   IF #AOn THEN GOTO MISC; END_IF;
END_REGION

REGION Network 149: No Local, Jump = TEST
   LOC:
   IF NOT #ModeLocal THEN GOTO TEST; END_IF;
END_REGION

REGION Network 150: State: Local - Not Active
   IF #CMD_QStop OR #FromStopState OR #FromStateAuto OR #FromStateManual THEN
       #BlockInfo.State_Act := 400;
   END_IF;
END_REGION

REGION Network 151: State: Local - Actiuve (Auto Start)
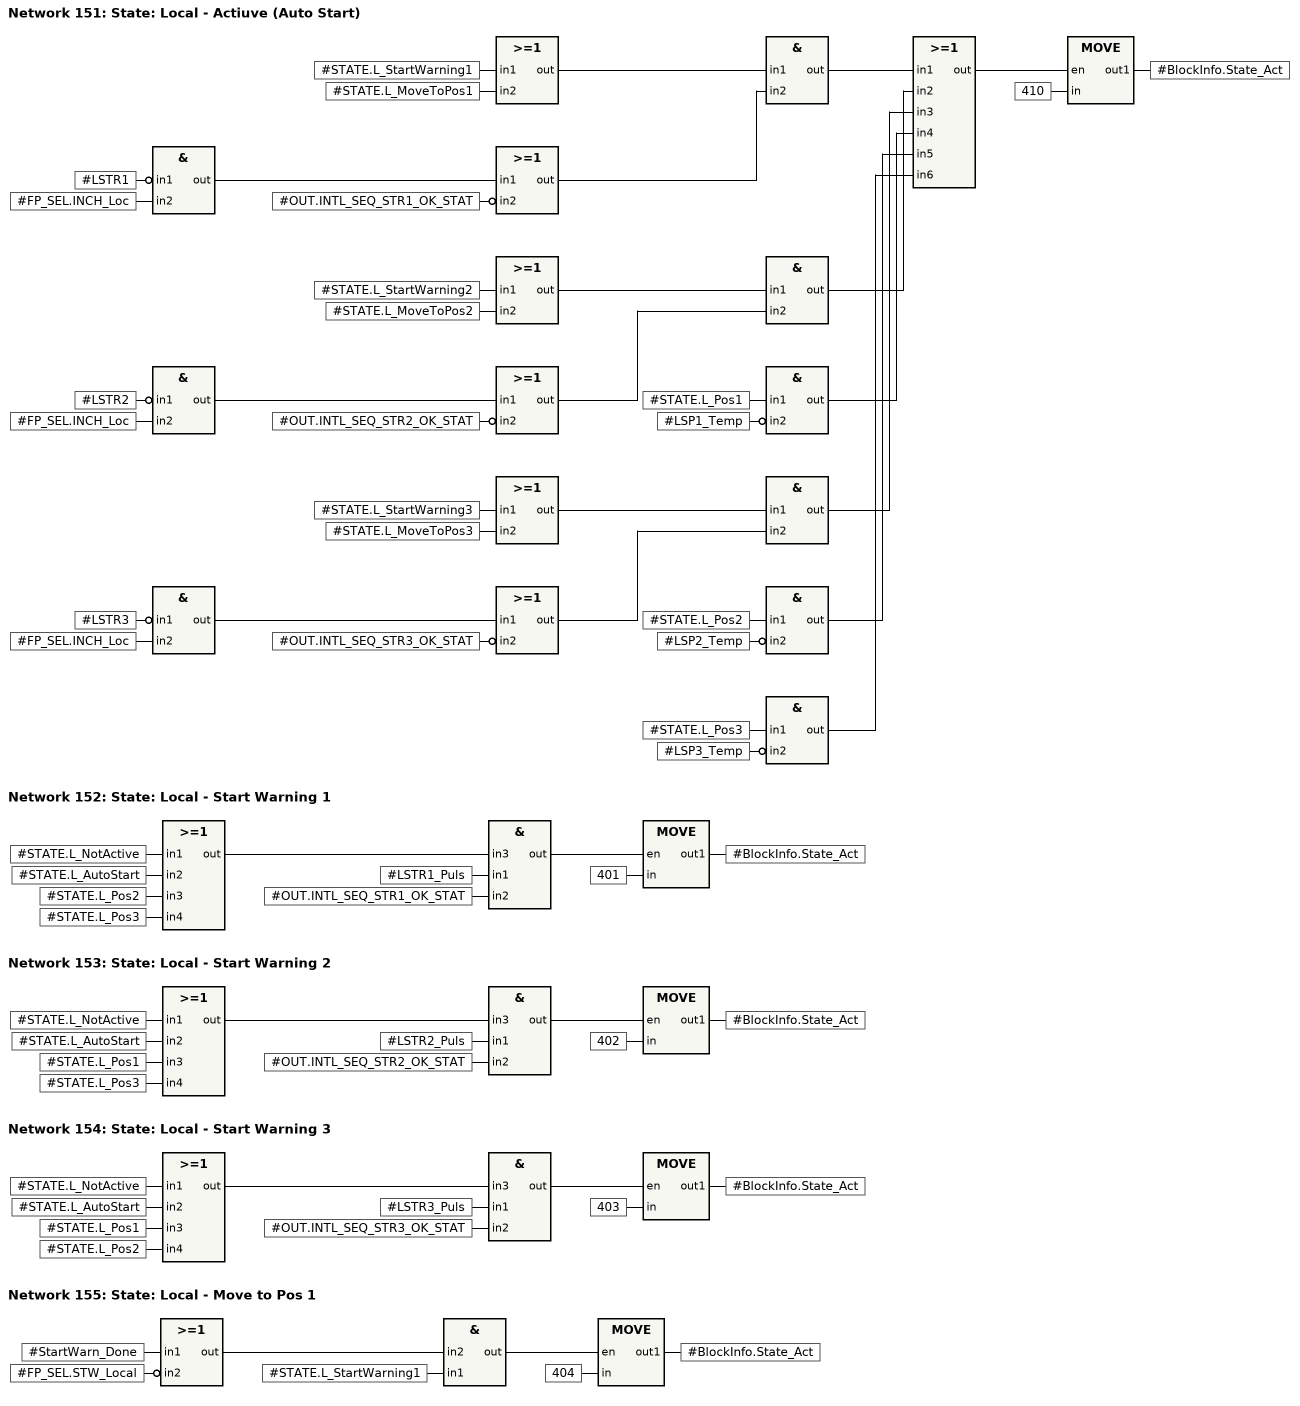
   IF ((#STATE.L_StartWarning1 OR #STATE.L_MoveToPos1) AND ((NOT #LSTR1 AND #FP_SEL.INCH_Loc) OR NOT #OUT.INTL_SEQ_STR1_OK_STAT)) OR ((#STATE.L_StartWarning2 OR #STATE.L_MoveToPos2) AND ((NOT #LSTR2 AND #FP_SEL.INCH_Loc) OR NOT #OUT.INTL_SEQ_STR2_OK_STAT)) OR ((#STATE.L_StartWarning3 OR #STATE.L_MoveToPos3) AND ((NOT #LSTR3 AND #FP_SEL.INCH_Loc) OR NOT #OUT.INTL_SEQ_STR3_OK_STAT)) OR (#STATE.L_Pos1 AND NOT #LSP1_Temp) OR (#STATE.L_Pos2 AND NOT #LSP2_Temp) OR (#STATE.L_Pos3 AND NOT #LSP3_Temp) THEN
       #BlockInfo.State_Act := 410;
   END_IF;
END_REGION

REGION Network 152: State: Local - Start Warning 1
   IF (#STATE.L_NotActive OR #STATE.L_AutoStart OR #STATE.L_Pos2 OR #STATE.L_Pos3) AND #LSTR1_Puls AND #OUT.INTL_SEQ_STR1_OK_STAT THEN
       #BlockInfo.State_Act := 401;
   END_IF;
END_REGION

REGION Network 153: State: Local - Start Warning 2
   IF (#STATE.L_NotActive OR #STATE.L_AutoStart OR #STATE.L_Pos1 OR #STATE.L_Pos3) AND #LSTR2_Puls AND #OUT.INTL_SEQ_STR2_OK_STAT THEN
       #BlockInfo.State_Act := 402;
   END_IF;
END_REGION

REGION Network 154: State: Local - Start Warning 3
   IF (#STATE.L_NotActive OR #STATE.L_AutoStart OR #STATE.L_Pos1 OR #STATE.L_Pos2) AND #LSTR3_Puls AND #OUT.INTL_SEQ_STR3_OK_STAT THEN
       #BlockInfo.State_Act := 403;
   END_IF;
END_REGION

REGION Network 155: State: Local - Move to Pos 1
   IF (#StartWarn_Done OR NOT #FP_SEL.STW_Local) AND #STATE.L_StartWarning1 THEN
       #BlockInfo.State_Act := 404;
   END_IF;
END_REGION

REGION Network 156: State: Local - Move to Pos 2
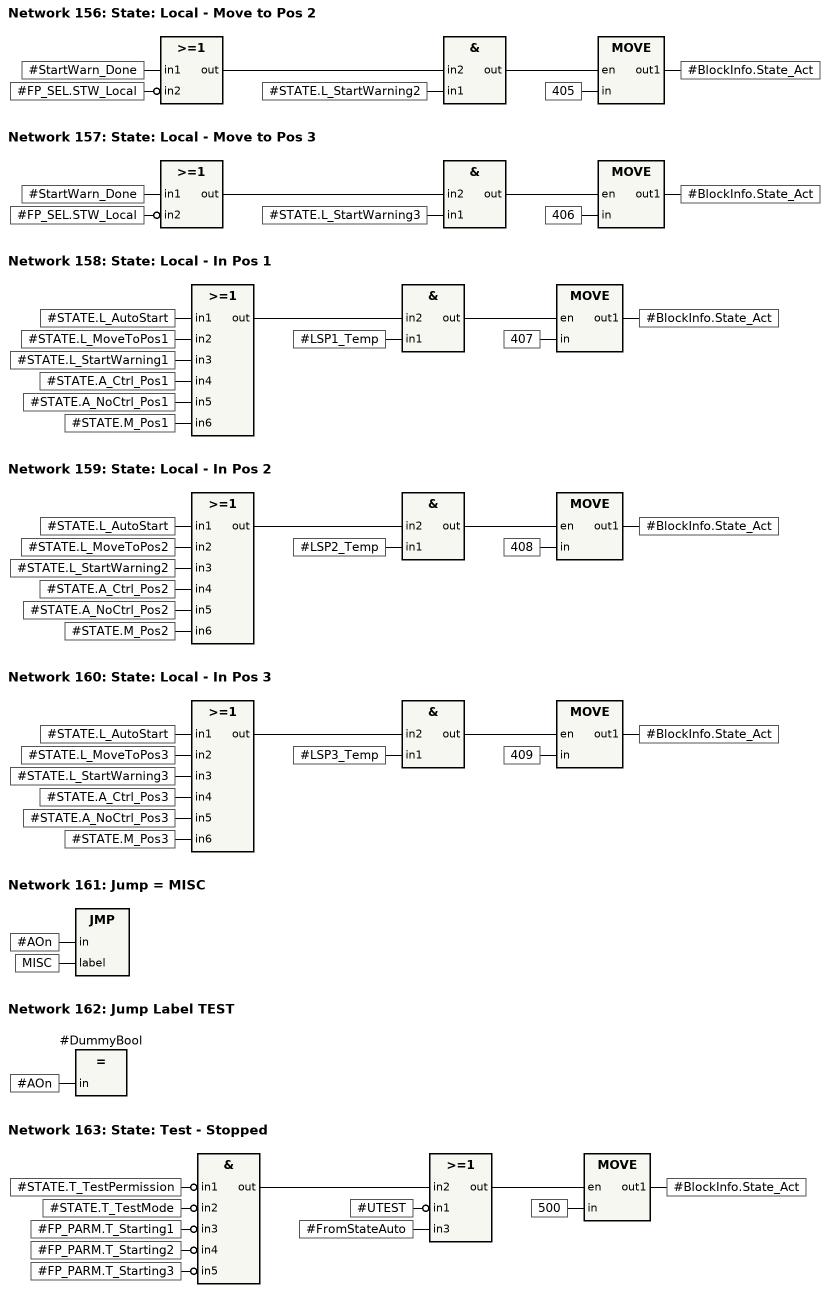
   IF (#StartWarn_Done OR NOT #FP_SEL.STW_Local) AND #STATE.L_StartWarning2 THEN
       #BlockInfo.State_Act := 405;
   END_IF;
END_REGION

REGION Network 157: State: Local - Move to Pos 3
   IF (#StartWarn_Done OR NOT #FP_SEL.STW_Local) AND #STATE.L_StartWarning3 THEN
       #BlockInfo.State_Act := 406;
   END_IF;
END_REGION

REGION Network 158: State: Local - In Pos 1
   IF (#STATE.L_AutoStart OR #STATE.L_MoveToPos1 OR #STATE.L_StartWarning1 OR #STATE.A_Ctrl_Pos1 OR #STATE.A_NoCtrl_Pos1 OR #STATE.M_Pos1) AND #LSP1_Temp THEN
       #BlockInfo.State_Act := 407;
   END_IF;
END_REGION

REGION Network 159: State: Local - In Pos 2
   IF (#STATE.L_AutoStart OR #STATE.L_MoveToPos2 OR #STATE.L_StartWarning2 OR #STATE.A_Ctrl_Pos2 OR #STATE.A_NoCtrl_Pos2 OR #STATE.M_Pos2) AND #LSP2_Temp THEN
       #BlockInfo.State_Act := 408;
   END_IF;
END_REGION

REGION Network 160: State: Local - In Pos 3
   IF (#STATE.L_AutoStart OR #STATE.L_MoveToPos3 OR #STATE.L_StartWarning3 OR #STATE.A_Ctrl_Pos3 OR #STATE.A_NoCtrl_Pos3 OR #STATE.M_Pos3) AND #LSP3_Temp THEN
       #BlockInfo.State_Act := 409;
   END_IF;
END_REGION

REGION Network 161: Jump = MISC
   IF #AOn THEN GOTO MISC; END_IF;
END_REGION

REGION Network 162: Jump Label TEST
   TEST:
   #DummyBool := #AOn;
END_REGION

REGION Network 163: State: Test - Stopped
   IF (NOT #STATE.T_TestPermission AND NOT #STATE.T_TestMode AND NOT #FP_PARM.T_Starting1 AND NOT #FP_PARM.T_Starting2 AND NOT #FP_PARM.T_Starting3) OR NOT #UTEST OR #FromStateAuto THEN
       #BlockInfo.State_Act := 500;
   END_IF;
END_REGION

REGION Network 164: State: Test - Test Mode
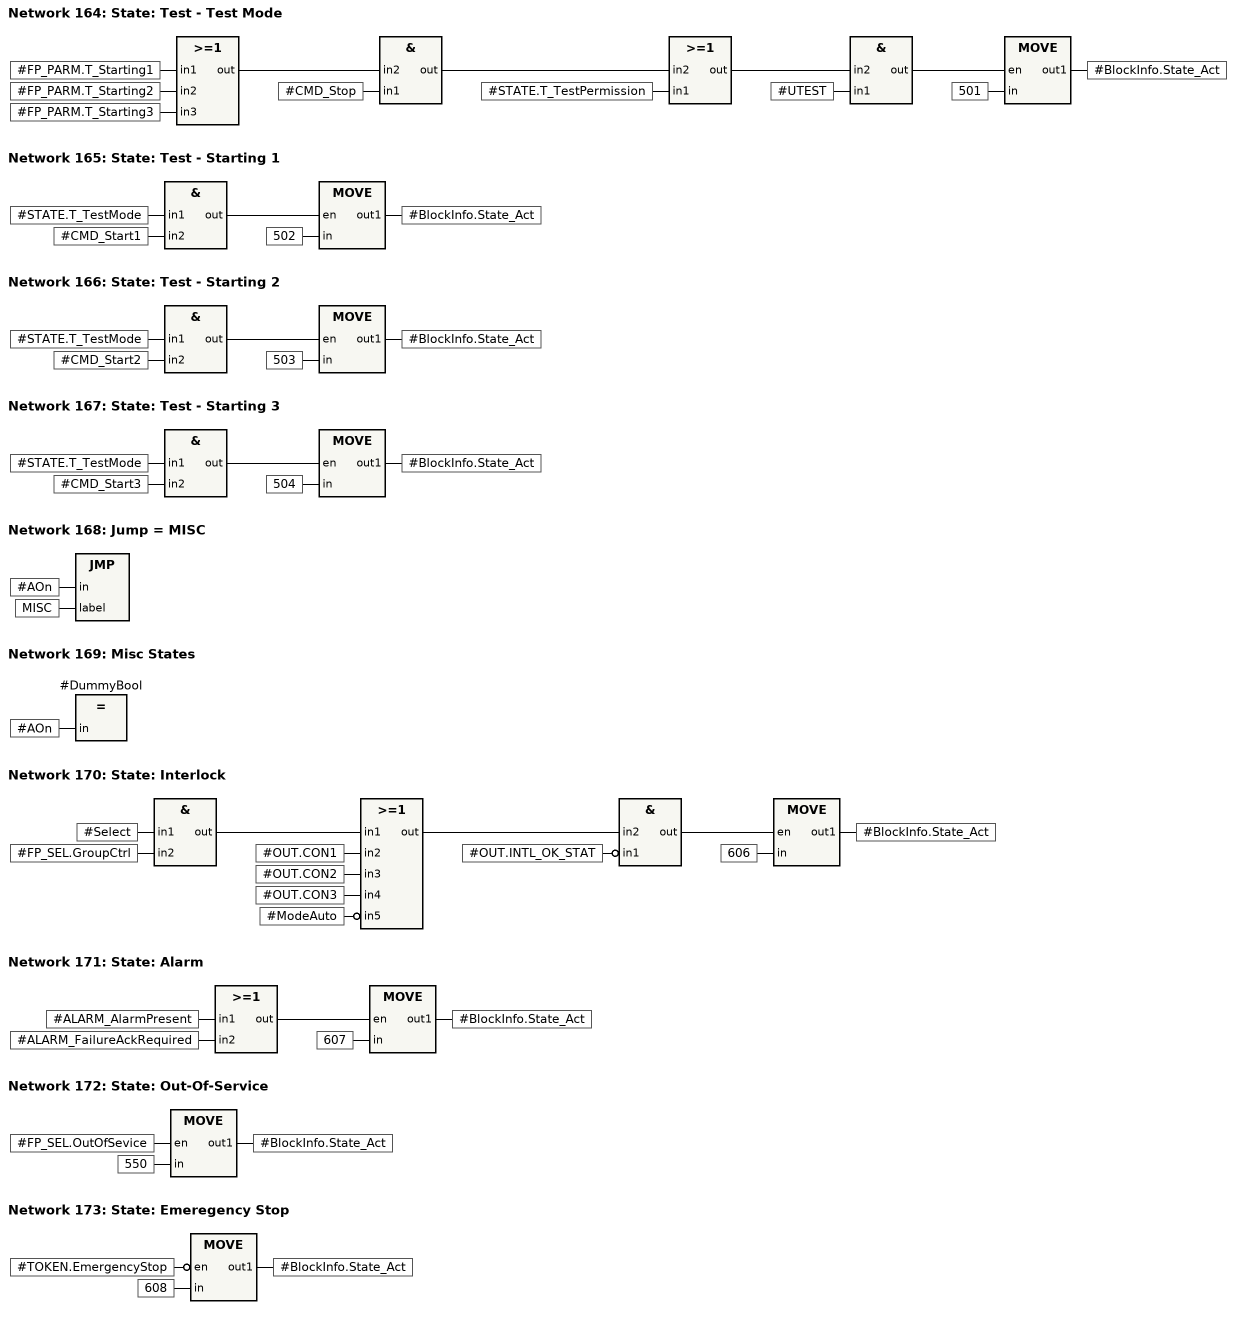
   IF (((#FP_PARM.T_Starting1 OR #FP_PARM.T_Starting2 OR #FP_PARM.T_Starting3) AND #CMD_Stop) OR #STATE.T_TestPermission) AND #UTEST THEN
       #BlockInfo.State_Act := 501;
   END_IF;
END_REGION

REGION Network 165: State: Test - Starting 1
   IF #STATE.T_TestMode AND #CMD_Start1 THEN #BlockInfo.State_Act := 502; END_IF;
END_REGION

REGION Network 166: State: Test - Starting 2
   IF #STATE.T_TestMode AND #CMD_Start2 THEN #BlockInfo.State_Act := 503; END_IF;
END_REGION

REGION Network 167: State: Test - Starting 3
   IF #STATE.T_TestMode AND #CMD_Start3 THEN #BlockInfo.State_Act := 504; END_IF;
END_REGION

REGION Network 168: Jump = MISC
   IF #AOn THEN GOTO MISC; END_IF;
END_REGION

REGION Network 169: Misc States
   MISC:
   #DummyBool := #AOn;
END_REGION

REGION Network 170: State: Interlock
   IF ((#Select AND #FP_SEL.GroupCtrl) OR #OUT.CON1 OR #OUT.CON2 OR #OUT.CON3 OR NOT #ModeAuto) AND NOT #OUT.INTL_OK_STAT THEN
       #BlockInfo.State_Act := 606;
   END_IF;
END_REGION

REGION Network 171: State: Alarm
   IF #ALARM_AlarmPresent OR #ALARM_FailureAckRequired THEN #BlockInfo.State_Act := 607; END_IF;
END_REGION

REGION Network 172: State: Out-Of-Service
   IF #FP_SEL.OutOfSevice THEN #BlockInfo.State_Act := 550; END_IF;
END_REGION

REGION Network 173: State: Emeregency Stop
   IF NOT #TOKEN.EmergencyStop THEN #BlockInfo.State_Act := 608; END_IF;
END_REGION

REGION Network 174: Reset Command Flag Before State Set - CON1
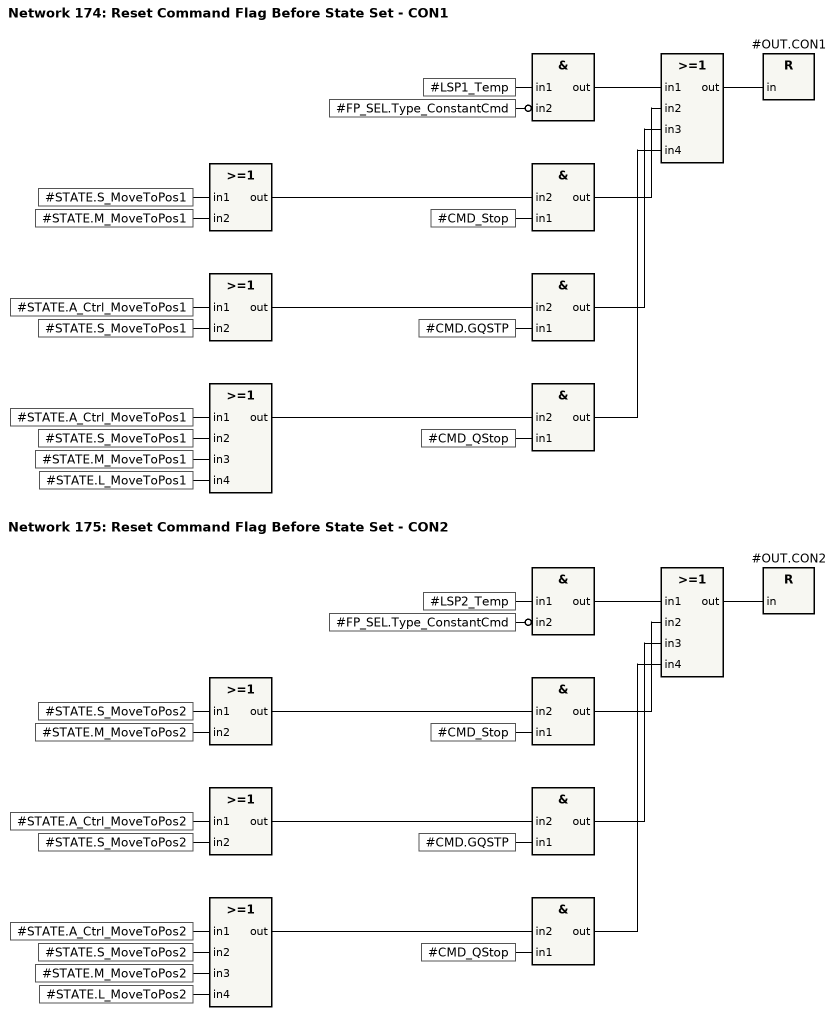
   IF (#LSP1_Temp AND NOT #FP_SEL.Type_ConstantCmd) OR ((#STATE.S_MoveToPos1 OR #STATE.M_MoveToPos1) AND #CMD_Stop) OR ((#STATE.A_Ctrl_MoveToPos1 OR #STATE.S_MoveToPos1) AND #CMD.GQSTP) OR ((#STATE.A_Ctrl_MoveToPos1 OR #STATE.S_MoveToPos1 OR #STATE.M_MoveToPos1 OR #STATE.L_MoveToPos1) AND #CMD_QStop) THEN
       #OUT.CON1 := FALSE;
   END_IF;
END_REGION

REGION Network 175: Reset Command Flag Before State Set - CON2
   IF (#LSP2_Temp AND NOT #FP_SEL.Type_ConstantCmd) OR ((#STATE.S_MoveToPos2 OR #STATE.M_MoveToPos2) AND #CMD_Stop) OR ((#STATE.A_Ctrl_MoveToPos2 OR #STATE.S_MoveToPos2) AND #CMD.GQSTP) OR ((#STATE.A_Ctrl_MoveToPos2 OR #STATE.S_MoveToPos2 OR #STATE.M_MoveToPos2 OR #STATE.L_MoveToPos2) AND #CMD_QStop) THEN
       #OUT.CON2 := FALSE;
   END_IF;
END_REGION

REGION Network 176: Reset Command Flag Before State Set - CON3
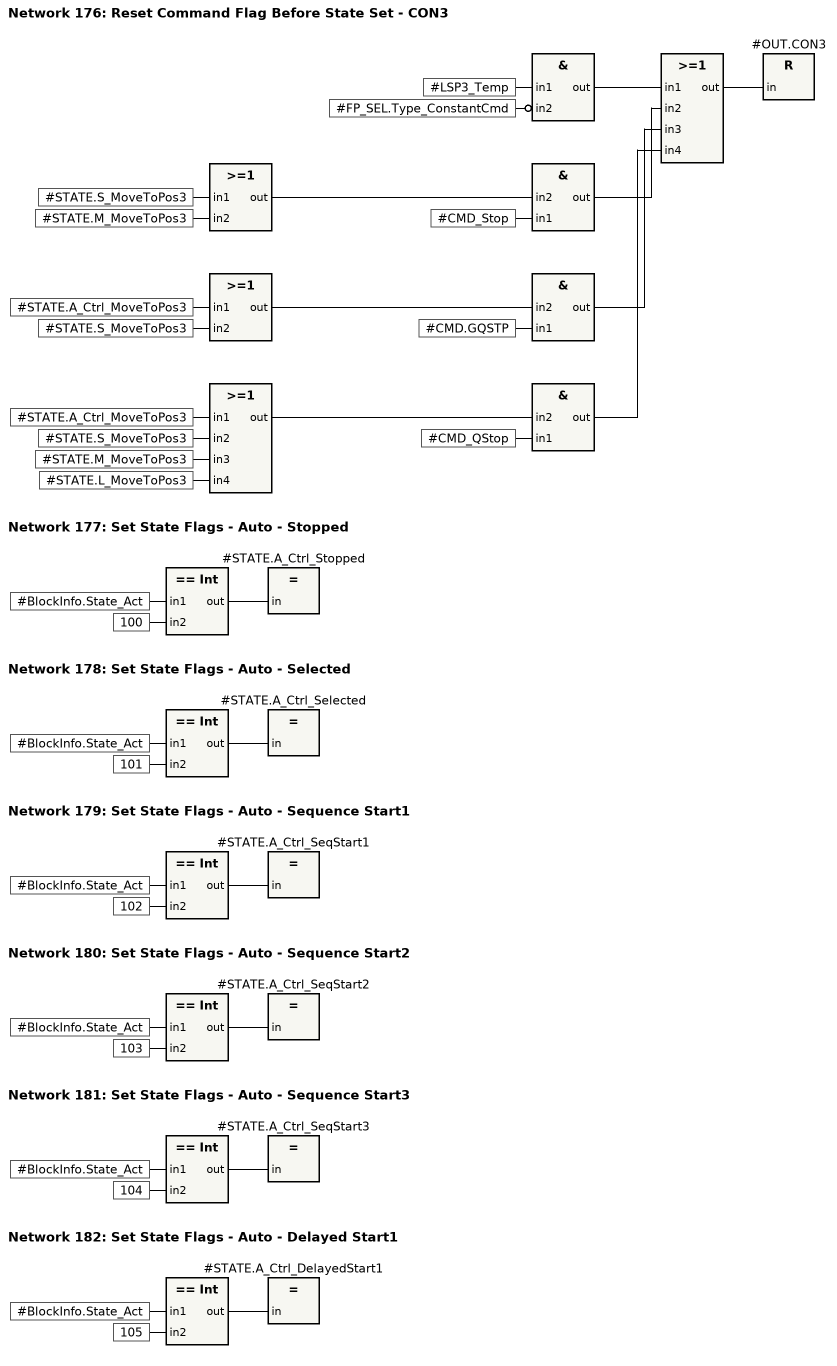
   IF (#LSP3_Temp AND NOT #FP_SEL.Type_ConstantCmd) OR ((#STATE.S_MoveToPos3 OR #STATE.M_MoveToPos3) AND #CMD_Stop) OR ((#STATE.A_Ctrl_MoveToPos3 OR #STATE.S_MoveToPos3) AND #CMD.GQSTP) OR ((#STATE.A_Ctrl_MoveToPos3 OR #STATE.S_MoveToPos3 OR #STATE.M_MoveToPos3 OR #STATE.L_MoveToPos3) AND #CMD_QStop) THEN
       #OUT.CON3 := FALSE;
   END_IF;
END_REGION

REGION Network 177: Set State Flags - Auto - Stopped
   #STATE.A_Ctrl_Stopped := #BlockInfo.State_Act = 100;
END_REGION

REGION Network 178: Set State Flags - Auto - Selected
   #STATE.A_Ctrl_Selected := #BlockInfo.State_Act = 101;
END_REGION

REGION Network 179: Set State Flags - Auto - Sequence Start1
   #STATE.A_Ctrl_SeqStart1 := #BlockInfo.State_Act = 102;
END_REGION

REGION Network 180: Set State Flags - Auto - Sequence Start2
   #STATE.A_Ctrl_SeqStart2 := #BlockInfo.State_Act = 103;
END_REGION

REGION Network 181: Set State Flags - Auto - Sequence Start3
   #STATE.A_Ctrl_SeqStart3 := #BlockInfo.State_Act = 104;
END_REGION

REGION Network 182: Set State Flags - Auto - Delayed Start1
   #STATE.A_Ctrl_DelayedStart1 := #BlockInfo.State_Act = 105;
END_REGION

REGION Network 183: Set State Flags - Auto - Delayed Start2
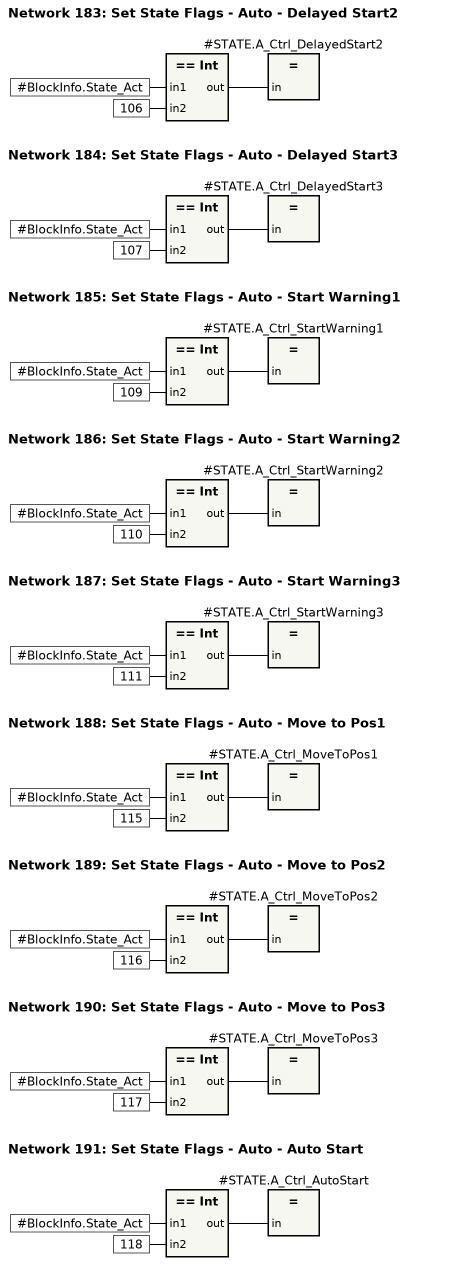
   #STATE.A_Ctrl_DelayedStart2 := #BlockInfo.State_Act = 106;
END_REGION

REGION Network 184: Set State Flags - Auto - Delayed Start3
   #STATE.A_Ctrl_DelayedStart3 := #BlockInfo.State_Act = 107;
END_REGION

REGION Network 185: Set State Flags - Auto - Start Warning1
   #STATE.A_Ctrl_StartWarning1 := #BlockInfo.State_Act = 109;
END_REGION

REGION Network 186: Set State Flags - Auto - Start Warning2
   #STATE.A_Ctrl_StartWarning2 := #BlockInfo.State_Act = 110;
END_REGION

REGION Network 187: Set State Flags - Auto - Start Warning3
   #STATE.A_Ctrl_StartWarning3 := #BlockInfo.State_Act = 111;
END_REGION

REGION Network 188: Set State Flags - Auto - Move to Pos1
   #STATE.A_Ctrl_MoveToPos1 := #BlockInfo.State_Act = 115;
END_REGION

REGION Network 189: Set State Flags - Auto - Move to Pos2
   #STATE.A_Ctrl_MoveToPos2 := #BlockInfo.State_Act = 116;
END_REGION

REGION Network 190: Set State Flags - Auto - Move to Pos3
   #STATE.A_Ctrl_MoveToPos3 := #BlockInfo.State_Act = 117;
END_REGION

REGION Network 191: Set State Flags - Auto - Auto Start
   #STATE.A_Ctrl_AutoStart := #BlockInfo.State_Act = 118;
END_REGION

REGION Network 192: Set State Flags - Auto - Position1
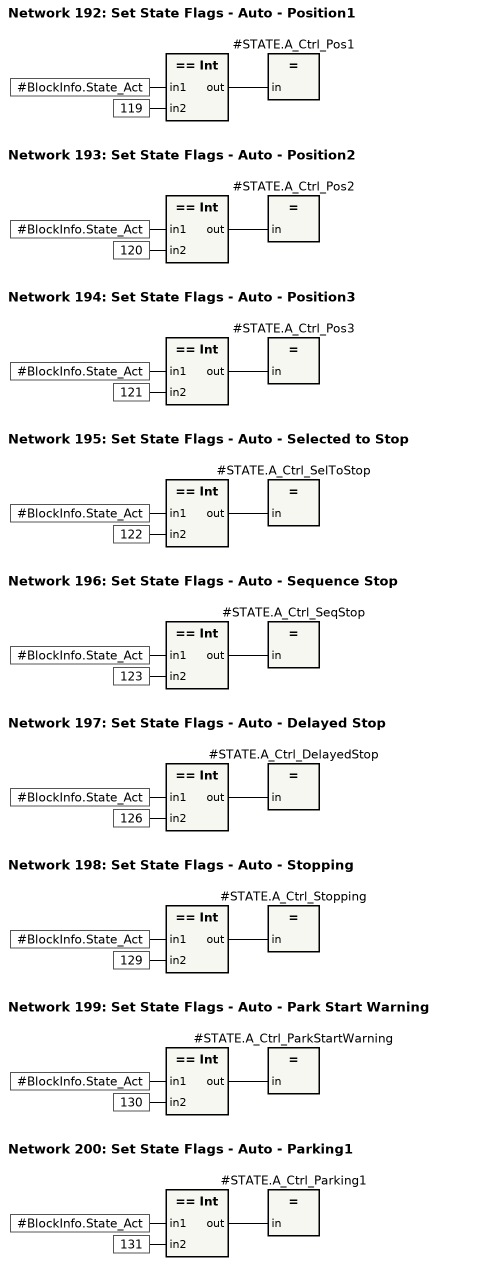
   #STATE.A_Ctrl_Pos1 := #BlockInfo.State_Act = 119;
END_REGION

REGION Network 193: Set State Flags - Auto - Position2
   #STATE.A_Ctrl_Pos2 := #BlockInfo.State_Act = 120;
END_REGION

REGION Network 194: Set State Flags - Auto - Position3
   #STATE.A_Ctrl_Pos3 := #BlockInfo.State_Act = 121;
END_REGION

REGION Network 195: Set State Flags - Auto - Selected to Stop
   #STATE.A_Ctrl_SelToStop := #BlockInfo.State_Act = 122;
END_REGION

REGION Network 196: Set State Flags - Auto - Sequence Stop
   #STATE.A_Ctrl_SeqStop := #BlockInfo.State_Act = 123;
END_REGION

REGION Network 197: Set State Flags - Auto - Delayed Stop
   #STATE.A_Ctrl_DelayedStop := #BlockInfo.State_Act = 126;
END_REGION

REGION Network 198: Set State Flags - Auto - Stopping
   #STATE.A_Ctrl_Stopping := #BlockInfo.State_Act = 129;
END_REGION

REGION Network 199: Set State Flags - Auto - Park Start Warning
   #STATE.A_Ctrl_ParkStartWarning := #BlockInfo.State_Act = 130;
END_REGION

REGION Network 200: Set State Flags - Auto - Parking1
   #STATE.A_Ctrl_Parking1 := #BlockInfo.State_Act = 131;
END_REGION

REGION Network 201: Set State Flags - Auto - Parking2
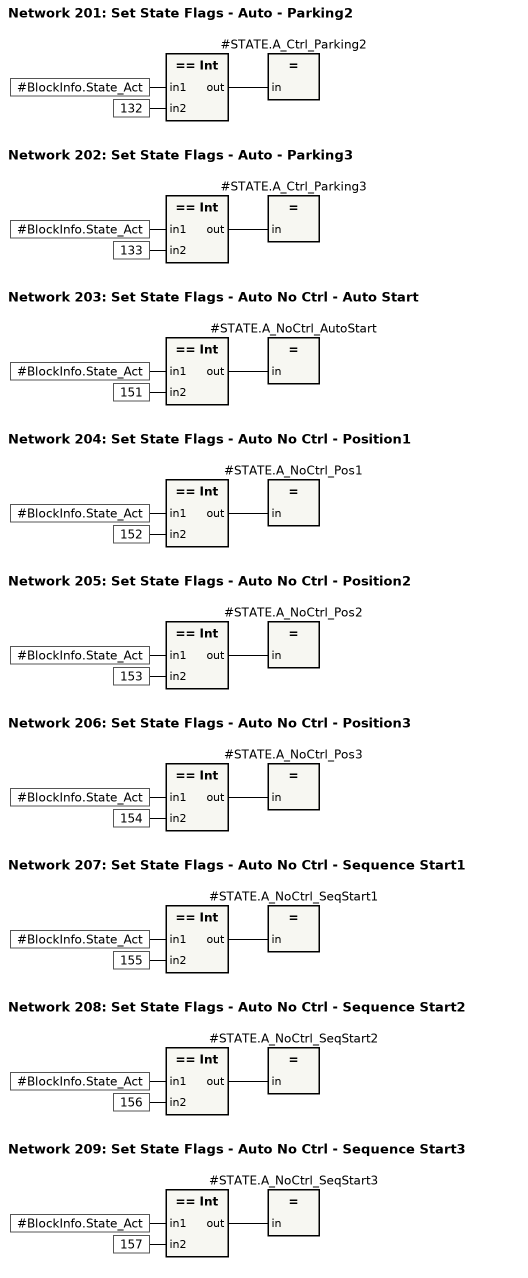
   #STATE.A_Ctrl_Parking2 := #BlockInfo.State_Act = 132;
END_REGION

REGION Network 202: Set State Flags - Auto - Parking3
   #STATE.A_Ctrl_Parking3 := #BlockInfo.State_Act = 133;
END_REGION

REGION Network 203: Set State Flags - Auto No Ctrl - Auto Start
   #STATE.A_NoCtrl_AutoStart := #BlockInfo.State_Act = 151;
END_REGION

REGION Network 204: Set State Flags - Auto No Ctrl - Position1
   #STATE.A_NoCtrl_Pos1 := #BlockInfo.State_Act = 152;
END_REGION

REGION Network 205: Set State Flags - Auto No Ctrl - Position2
   #STATE.A_NoCtrl_Pos2 := #BlockInfo.State_Act = 153;
END_REGION

REGION Network 206: Set State Flags - Auto No Ctrl - Position3
   #STATE.A_NoCtrl_Pos3 := #BlockInfo.State_Act = 154;
END_REGION

REGION Network 207: Set State Flags - Auto No Ctrl - Sequence Start1
   #STATE.A_NoCtrl_SeqStart1 := #BlockInfo.State_Act = 155;
END_REGION

REGION Network 208: Set State Flags - Auto No Ctrl - Sequence Start2
   #STATE.A_NoCtrl_SeqStart2 := #BlockInfo.State_Act = 156;
END_REGION

REGION Network 209: Set State Flags - Auto No Ctrl - Sequence Start3
   #STATE.A_NoCtrl_SeqStart3 := #BlockInfo.State_Act = 157;
END_REGION

REGION Network 210: Set State Flags - Auto No Ctrl - Start Warning1
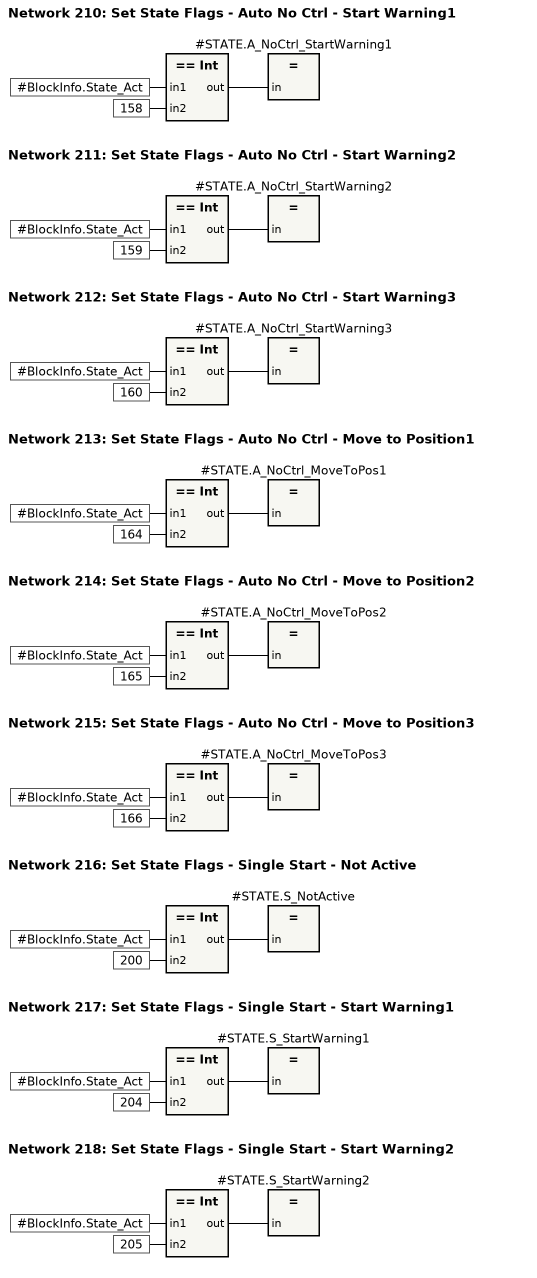
   #STATE.A_NoCtrl_StartWarning1 := #BlockInfo.State_Act = 158;
END_REGION

REGION Network 211: Set State Flags - Auto No Ctrl - Start Warning2
   #STATE.A_NoCtrl_StartWarning2 := #BlockInfo.State_Act = 159;
END_REGION

REGION Network 212: Set State Flags - Auto No Ctrl - Start Warning3
   #STATE.A_NoCtrl_StartWarning3 := #BlockInfo.State_Act = 160;
END_REGION

REGION Network 213: Set State Flags - Auto No Ctrl - Move to Position1
   #STATE.A_NoCtrl_MoveToPos1 := #BlockInfo.State_Act = 164;
END_REGION

REGION Network 214: Set State Flags - Auto No Ctrl - Move to Position2
   #STATE.A_NoCtrl_MoveToPos2 := #BlockInfo.State_Act = 165;
END_REGION

REGION Network 215: Set State Flags - Auto No Ctrl - Move to Position3
   #STATE.A_NoCtrl_MoveToPos3 := #BlockInfo.State_Act = 166;
END_REGION

REGION Network 216: Set State Flags - Single Start - Not Active
   #STATE.S_NotActive := #BlockInfo.State_Act = 200;
END_REGION

REGION Network 217: Set State Flags - Single Start - Start Warning1
   #STATE.S_StartWarning1 := #BlockInfo.State_Act = 204;
END_REGION

REGION Network 218: Set State Flags - Single Start - Start Warning2
   #STATE.S_StartWarning2 := #BlockInfo.State_Act = 205;
END_REGION

REGION Network 219: Set State Flags - Single Start - Start Warning3
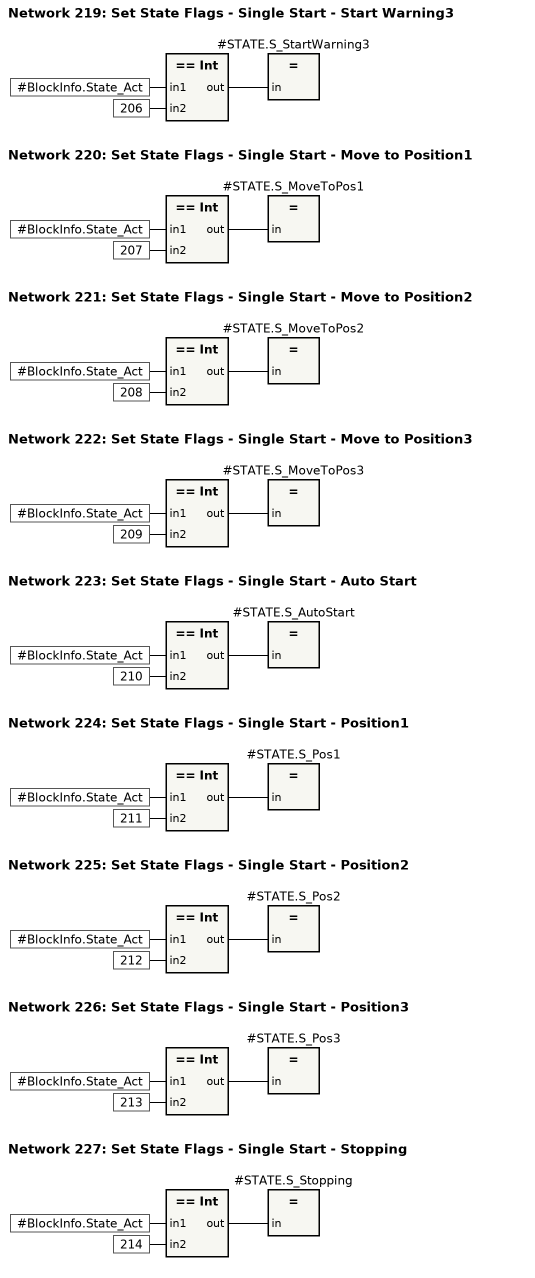
   #STATE.S_StartWarning3 := #BlockInfo.State_Act = 206;
END_REGION

REGION Network 220: Set State Flags - Single Start - Move to Position1
   #STATE.S_MoveToPos1 := #BlockInfo.State_Act = 207;
END_REGION

REGION Network 221: Set State Flags - Single Start - Move to Position2
   #STATE.S_MoveToPos2 := #BlockInfo.State_Act = 208;
END_REGION

REGION Network 222: Set State Flags - Single Start - Move to Position3
   #STATE.S_MoveToPos3 := #BlockInfo.State_Act = 209;
END_REGION

REGION Network 223: Set State Flags - Single Start - Auto Start
   #STATE.S_AutoStart := #BlockInfo.State_Act = 210;
END_REGION

REGION Network 224: Set State Flags - Single Start - Position1
   #STATE.S_Pos1 := #BlockInfo.State_Act = 211;
END_REGION

REGION Network 225: Set State Flags - Single Start - Position2
   #STATE.S_Pos2 := #BlockInfo.State_Act = 212;
END_REGION

REGION Network 226: Set State Flags - Single Start - Position3
   #STATE.S_Pos3 := #BlockInfo.State_Act = 213;
END_REGION

REGION Network 227: Set State Flags - Single Start - Stopping
   #STATE.S_Stopping := #BlockInfo.State_Act = 214;
END_REGION

REGION Network 228: Set State Flags - Single Start - Park Start Warning
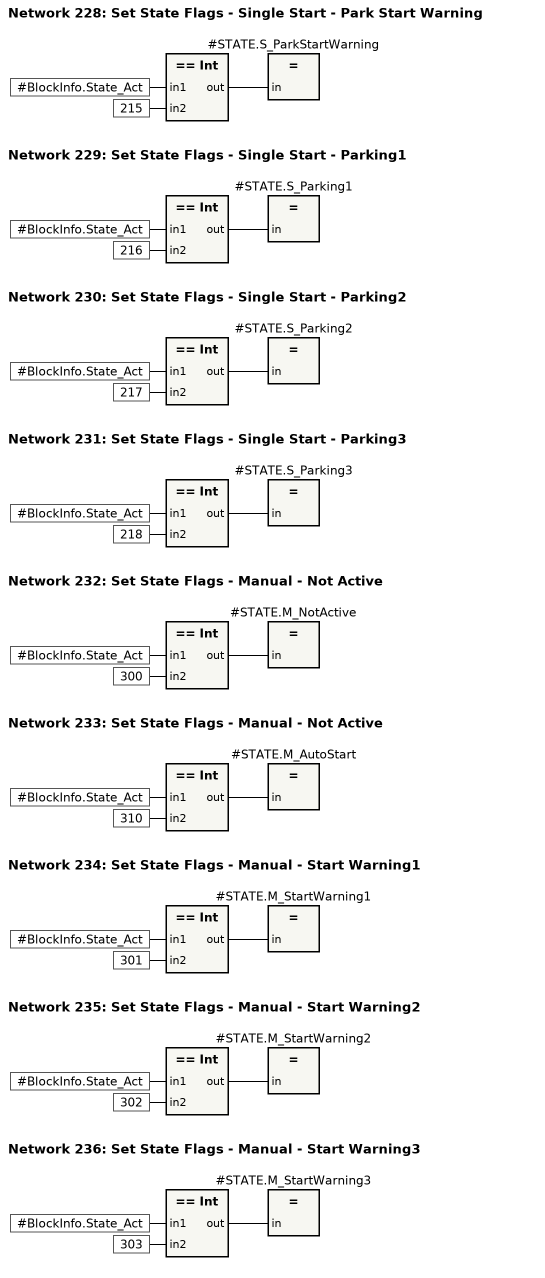
   #STATE.S_ParkStartWarning := #BlockInfo.State_Act = 215;
END_REGION

REGION Network 229: Set State Flags - Single Start - Parking1
   #STATE.S_Parking1 := #BlockInfo.State_Act = 216;
END_REGION

REGION Network 230: Set State Flags - Single Start - Parking2
   #STATE.S_Parking2 := #BlockInfo.State_Act = 217;
END_REGION

REGION Network 231: Set State Flags - Single Start - Parking3
   #STATE.S_Parking3 := #BlockInfo.State_Act = 218;
END_REGION

REGION Network 232: Set State Flags - Manual - Not Active
   #STATE.M_NotActive := #BlockInfo.State_Act = 300;
END_REGION

REGION Network 233: Set State Flags - Manual - Not Active
   #STATE.M_AutoStart := #BlockInfo.State_Act = 310;
END_REGION

REGION Network 234: Set State Flags - Manual - Start Warning1
   #STATE.M_StartWarning1 := #BlockInfo.State_Act = 301;
END_REGION

REGION Network 235: Set State Flags - Manual - Start Warning2
   #STATE.M_StartWarning2 := #BlockInfo.State_Act = 302;
END_REGION

REGION Network 236: Set State Flags - Manual - Start Warning3
   #STATE.M_StartWarning3 := #BlockInfo.State_Act = 303;
END_REGION

REGION Network 237: Set State Flags - Manual - Move to Position1
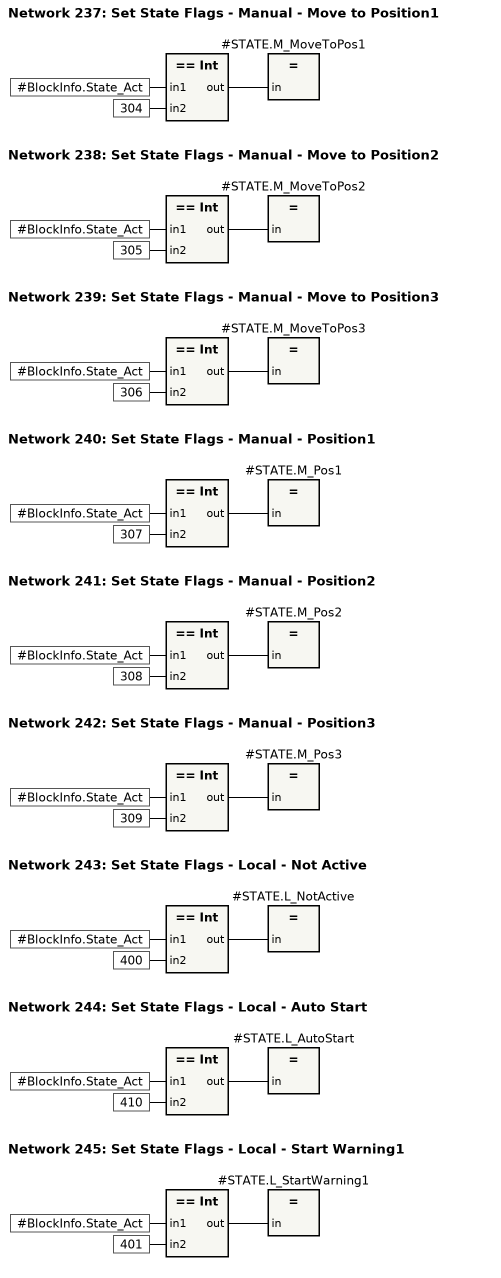
   #STATE.M_MoveToPos1 := #BlockInfo.State_Act = 304;
END_REGION

REGION Network 238: Set State Flags - Manual - Move to Position2
   #STATE.M_MoveToPos2 := #BlockInfo.State_Act = 305;
END_REGION

REGION Network 239: Set State Flags - Manual - Move to Position3
   #STATE.M_MoveToPos3 := #BlockInfo.State_Act = 306;
END_REGION

REGION Network 240: Set State Flags - Manual - Position1
   #STATE.M_Pos1 := #BlockInfo.State_Act = 307;
END_REGION

REGION Network 241: Set State Flags - Manual - Position2
   #STATE.M_Pos2 := #BlockInfo.State_Act = 308;
END_REGION

REGION Network 242: Set State Flags - Manual - Position3
   #STATE.M_Pos3 := #BlockInfo.State_Act = 309;
END_REGION

REGION Network 243: Set State Flags - Local - Not Active
   #STATE.L_NotActive := #BlockInfo.State_Act = 400;
END_REGION

REGION Network 244: Set State Flags - Local - Auto Start
   #STATE.L_AutoStart := #BlockInfo.State_Act = 410;
END_REGION

REGION Network 245: Set State Flags - Local - Start Warning1
   #STATE.L_StartWarning1 := #BlockInfo.State_Act = 401;
END_REGION

REGION Network 246: Set State Flags - Local - Start Warning2
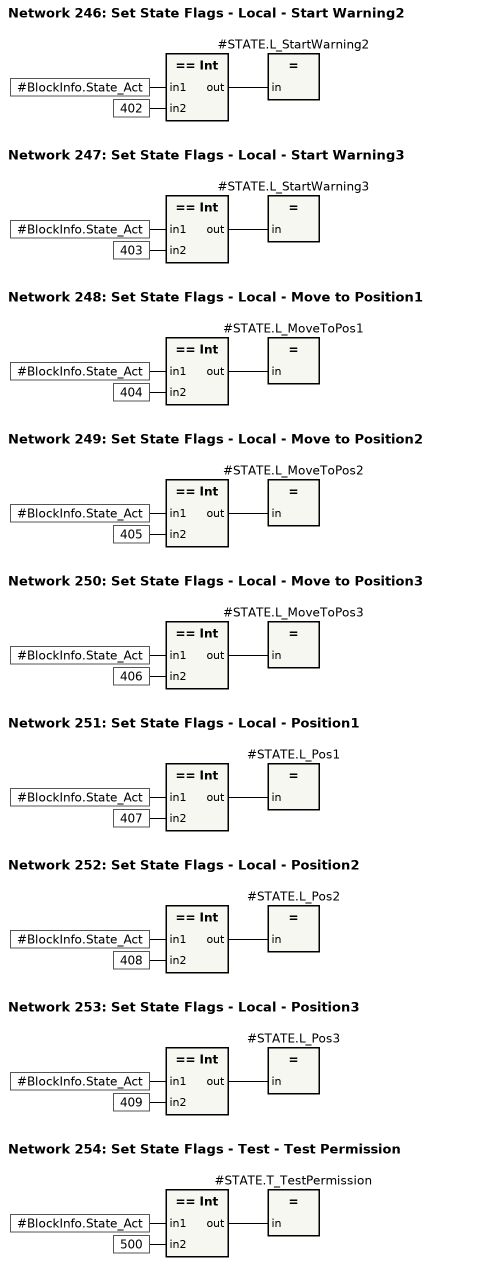
   #STATE.L_StartWarning2 := #BlockInfo.State_Act = 402;
END_REGION

REGION Network 247: Set State Flags - Local - Start Warning3
   #STATE.L_StartWarning3 := #BlockInfo.State_Act = 403;
END_REGION

REGION Network 248: Set State Flags - Local - Move to Position1
   #STATE.L_MoveToPos1 := #BlockInfo.State_Act = 404;
END_REGION

REGION Network 249: Set State Flags - Local - Move to Position2
   #STATE.L_MoveToPos2 := #BlockInfo.State_Act = 405;
END_REGION

REGION Network 250: Set State Flags - Local - Move to Position3
   #STATE.L_MoveToPos3 := #BlockInfo.State_Act = 406;
END_REGION

REGION Network 251: Set State Flags - Local - Position1
   #STATE.L_Pos1 := #BlockInfo.State_Act = 407;
END_REGION

REGION Network 252: Set State Flags - Local - Position2
   #STATE.L_Pos2 := #BlockInfo.State_Act = 408;
END_REGION

REGION Network 253: Set State Flags - Local - Position3
   #STATE.L_Pos3 := #BlockInfo.State_Act = 409;
END_REGION

REGION Network 254: Set State Flags - Test - Test Permission
   #STATE.T_TestPermission := #BlockInfo.State_Act = 500;
END_REGION

REGION Network 255: Set State Flags - Test - Test Mode
